C08939=1021.076,209.738,-122.791,168.989,49.902,159.469
C08940=1021.082,209.986,-122.816,168.993,49.896,159.468
C08941=1021.088,210.234,-122.842,168.996,49.891,159.468
C08942=1021.094,210.483,-122.868,169.000,49.886,159.467
C08943=1021.100,210.732,-122.894,169.003,49.880,159.467
C08944=1021.107,210.980,-122.920,169.007,49.875,159.466
C08945=1021.112,211.229,-122.946,169.010,49.869,159.465
C08946=1021.118,211.478,-122.971,169.014,49.864,159.465
C08947=1021.125,211.726,-122.997,169.017,49.858,159.464
C08948=1021.130,211.975,-123.023,169.021,49.853,159.464
C08949=1021.137,212.223,-123.049,169.024,49.848,159.463
C08950=1021.143,212.471,-123.074,169.028,49.842,159.463
C08951=1021.149,212.721,-123.101,169.032,49.837,159.462
C08952=1021.156,212.969,-123.127,169.036,49.832,159.462
C08953=1021.162,213.218,-123.152,169.039,49.826,159.461
C08954=1021.168,213.466,-123.179,169.043,49.821,159.460
C08955=1021.174,213.715,-123.204,169.046,49.816,159.460
C08956=1021.180,213.963,-123.230,169.050,49.810,159.459
C08957=1021.186,214.212,-123.256,169.053,49.805,159.459
C08958=1021.193,214.461,-123.283,169.057,49.800,159.458
C08959=1021.199,214.709,-123.308,169.060,49.794,159.457
C08960=1021.206,214.957,-123.334,169.064,49.789,159.457
C08961=1021.211,215.206,-123.360,169.068,49.784,159.457
C08962=1021.218,215.454,-123.386,169.072,49.778,159.456
C08963=1021.224,215.704,-123.412,169.075,49.773,159.455
C08964=1021.230,215.952,-123.438,169.079,49.768,159.455
C08965=1021.236,216.201,-123.464,169.082,49.763,159.454
C08966=1021.243,216.449,-123.490,169.086,49.757,159.454
C08967=1021.248,216.698,-123.516,169.089,49.752,159.453
C08968=1021.255,216.946,-123.542,169.094,49.747,159.453
C08969=1021.262,217.194,-123.568,169.097,49.742,159.452
C08970=1021.267,217.443,-123.594,169.101,49.736,159.451
C08971=1021.274,217.692,-123.620,169.104,49.731,159.451
C08972=1021.281,217.941,-123.646,169.108,49.726,159.450
C08973=1021.287,218.189,-123.672,169.111,49.721,159.450
C08974=1021.293,218.437,-123.698,169.116,49.715,159.450
C08975=1021.299,218.686,-123.725,169.119,49.711,159.449
C08976=1021.304,218.905,-123.748,169.122,49.706,159.448
C08977=1021.310,219.125,-123.771,169.126,49.701,159.448
C08978=1021.315,219.343,-123.794,169.128,49.697,159.447
C08979=1021.321,219.562,-123.818,169.132,49.692,159.447
C08980=1021.326,219.782,-123.841,169.135,49.687,159.447
C08981=1021.332,220.001,-123.864,169.138,49.683,159.446
C08982=1021.337,220.221,-123.888,169.141,49.679,159.446
C08983=1021.342,220.439,-123.911,169.144,49.674,159.445
C08984=1021.349,220.688,-123.937,169.148,49.669,159.445
C08985=1021.355,220.937,-123.963,169.152,49.664,159.444
C08986=1021.361,221.185,-123.990,169.155,49.659,159.444
C08987=1021.367,221.433,-124.016,169.159,49.654,159.443
C08988=1021.373,221.682,-124.043,169.162,49.649,159.443
C08989=1021.379,221.931,-124.070,169.167,49.644,159.442
C08990=1021.386,222.179,-124.096,169.170,49.640,159.442
C08991=1021.392,222.428,-124.123,169.173,49.635,159.441
C08992=1021.399,222.676,-124.149,169.178,49.629,159.441
C08993=1021.404,222.925,-124.175,169.181,49.624,159.440
C08994=1021.410,223.174,-124.202,169.185,49.619,159.440
C08995=1021.417,223.422,-124.228,169.188,49.614,159.439
C08996=1021.423,223.670,-124.254,169.193,49.609,159.439
C08997=1021.429,223.919,-124.281,169.196,49.604,159.438
C08998=1021.436,224.167,-124.307,169.199,49.599,159.438
C08999=1021.442,224.416,-124.334,169.204,49.595,159.438
C09000=1021.448,224.665,-124.361,169.207,49.590,159.437
C09001=1021.454,224.913,-124.387,169.211,49.584,159.437
C09002=1021.461,225.162,-124.414,169.215,49.580,159.436
C09003=1021.467,225.410,-124.440,169.218,49.575,159.435
C09004=1021.473,225.658,-124.467,169.222,49.569,159.435
C09005=1021.479,225.907,-124.494,169.226,49.565,159.435
C09006=1021.486,226.155,-124.520,169.230,49.560,159.434
C09007=1021.492,226.404,-124.547,169.233,49.555,159.434
C09008=1021.498,226.653,-124.574,169.236,49.550,159.433
C09009=1021.505,226.901,-124.600,169.241,49.545,159.433
C09010=1021.511,227.149,-124.627,169.244,49.541,159.432
C09011=1021.517,227.398,-124.654,169.249,49.535,159.432
C09012=1021.523,227.647,-124.681,169.252,49.530,159.431
C09013=1021.529,227.895,-124.708,169.255,49.526,159.431
C09014=1021.535,228.144,-124.735,169.260,49.521,159.430
C09015=1021.542,228.392,-124.762,169.263,49.516,159.430
C09016=1021.548,228.640,-124.788,169.267,49.512,159.430
C09017=1021.554,228.889,-124.815,169.271,49.507,159.429
C09018=1021.560,229.137,-124.842,169.274,49.502,159.429
C09019=1021.567,229.386,-124.869,169.278,49.497,159.428
C09020=1021.573,229.634,-124.896,169.282,49.492,159.428
C09021=1021.579,229.883,-124.923,169.286,49.488,159.427
C09022=1021.585,230.131,-124.950,169.290,49.483,159.427
C09023=1021.592,230.380,-124.977,169.293,49.479,159.427
C09024=1021.597,230.628,-125.004,169.297,49.474,159.426
C09025=1021.604,230.877,-125.032,169.301,49.469,159.426
C09026=1021.610,231.125,-125.059,169.305,49.464,159.425
C09027=1021.616,231.374,-125.086,169.308,49.460,159.425
C09028=1021.622,231.622,-125.113,169.311,49.455,159.424
C09029=1021.629,231.871,-125.140,169.316,49.451,159.424
C09030=1021.635,232.119,-125.167,169.320,49.446,159.424
C09031=1021.641,232.368,-125.194,169.323,49.441,159.423
C09032=1021.647,232.616,-125.222,169.328,49.437,159.423
C09033=1021.653,232.865,-125.249,169.331,49.432,159.422
C09034=1021.660,233.112,-125.276,169.334,49.428,159.422
C09035=1021.666,233.361,-125.303,169.339,49.423,159.422
C09036=1021.671,233.576,-125.327,169.342,49.419,159.421
C09037=1021.677,233.792,-125.350,169.345,49.415,159.421
C09038=1021.682,234.007,-125.374,169.349,49.411,159.421
C09039=1021.687,234.222,-125.397,169.351,49.407,159.420
C09040=1021.693,234.437,-125.421,169.355,49.403,159.420
C09041=1021.698,234.652,-125.444,169.358,49.399,159.420
C09042=1021.704,234.867,-125.468,169.362,49.395,159.419
C09043=1021.709,235.083,-125.492,169.365,49.391,159.419
C09044=1021.715,235.330,-125.519,169.369,49.387,159.419
C09045=1021.722,235.579,-125.547,169.373,49.382,159.418
C09046=1021.728,235.828,-125.574,169.377,49.377,159.418
C09047=1021.734,236.076,-125.601,169.380,49.373,159.417
C09048=1021.740,236.325,-125.628,169.384,49.369,159.417
C09049=1021.747,236.573,-125.656,169.388,49.364,159.417
C09050=1021.753,236.821,-125.683,169.392,49.359,159.416
C09051=1021.760,237.070,-125.710,169.396,49.355,159.416
C09052=1021.765,237.318,-125.738,169.400,49.351,159.416
C09053=1021.772,237.566,-125.766,169.404,49.346,159.415
C09054=1021.778,237.816,-125.793,169.407,49.342,159.415
C09055=1021.784,238.063,-125.820,169.412,49.337,159.414
C09056=1021.791,238.312,-125.848,169.415,49.333,159.414
C09057=1021.797,238.561,-125.875,169.419,49.329,159.414
C09058=1021.803,238.809,-125.902,169.423,49.323,159.413
C09059=1021.810,239.057,-125.930,169.427,49.319,159.413
C09060=1021.816,239.306,-125.958,169.431,49.315,159.412
C09061=1021.822,239.553,-125.986,169.435,49.310,159.412
C09062=1021.828,239.803,-126.013,169.439,49.306,159.412
C09063=1021.834,240.051,-126.041,169.442,49.302,159.412
C09064=1021.840,240.299,-126.069,169.446,49.298,159.411
C09065=1021.847,240.547,-126.096,169.451,49.293,159.411
C09066=1021.853,240.796,-126.125,169.454,49.289,159.411
C09067=1021.859,241.044,-126.152,169.458,49.285,159.410
C09068=1021.865,241.293,-126.180,169.462,49.281,159.410
C09069=1021.872,241.541,-126.208,169.466,49.276,159.410
C09070=1021.878,241.790,-126.236,169.470,49.272,159.409
C09071=1021.884,242.038,-126.264,169.474,49.268,159.409
C09072=1021.890,242.286,-126.291,169.478,49.263,159.409
C09073=1021.897,242.535,-126.319,169.482,49.259,159.408
C09074=1021.903,242.783,-126.347,169.485,49.255,159.408
C09075=1021.909,243.031,-126.375,169.489,49.251,159.407
C09076=1021.915,243.280,-126.403,169.494,49.246,159.407
C09077=1021.922,243.528,-126.431,169.497,49.242,159.407
C09078=1021.927,243.776,-126.459,169.501,49.238,159.407
C09079=1021.934,244.025,-126.487,169.505,49.233,159.406
C09080=1021.940,244.273,-126.515,169.510,49.230,159.406
C09081=1021.946,244.522,-126.544,169.513,49.225,159.406
C09082=1021.952,244.769,-126.571,169.517,49.221,159.405
C09083=1021.958,245.018,-126.600,169.520,49.217,159.405
C09084=1021.964,245.267,-126.628,169.524,49.213,159.405
C09085=1021.970,245.515,-126.656,169.529,49.209,159.405
C09086=1021.976,245.763,-126.684,169.533,49.205,159.404
C09087=1021.982,246.011,-126.713,169.536,49.200,159.404
C09088=1021.989,246.260,-126.740,169.540,49.197,159.404
C09089=1021.995,246.509,-126.769,169.545,49.192,159.403
C09090=1022.001,246.757,-126.798,169.549,49.188,159.403
C09091=1022.007,247.004,-126.825,169.553,49.185,159.403
C09092=1022.013,247.253,-126.853,169.556,49.180,159.403
C09093=1022.019,247.501,-126.883,169.561,49.176,159.402
C09094=1022.026,247.750,-126.910,169.565,49.172,159.402
C09095=1022.032,247.999,-126.939,169.569,49.168,159.402
C09096=1022.037,248.210,-126.963,169.572,49.165,159.401
C09097=1022.042,248.423,-126.987,169.576,49.161,159.401
C09098=1022.048,248.634,-127.011,169.579,49.158,159.401
C09099=1022.053,248.847,-127.036,169.583,49.155,159.401
C09100=1022.058,249.058,-127.060,169.585,49.151,159.400
C09101=1022.064,249.270,-127.084,169.589,49.147,159.400
C09102=1022.069,249.482,-127.108,169.592,49.144,159.400
C09103=1022.074,249.694,-127.132,169.596,49.141,159.400
C09104=1022.080,249.942,-127.161,169.600,49.137,159.400
C09105=1022.087,250.191,-127.190,169.604,49.133,159.399
C09106=1022.093,250.439,-127.217,169.608,49.128,159.399
C09107=1022.099,250.687,-127.246,169.612,49.125,159.399
C09108=1022.105,250.936,-127.275,169.616,49.121,159.399
C09109=1022.112,251.184,-127.303,169.620,49.117,159.398
C09110=1022.118,251.432,-127.331,169.624,49.113,159.398
C09111=1022.125,251.681,-127.361,169.629,49.109,159.398
C09112=1022.131,251.929,-127.388,169.632,49.105,159.398
C09113=1022.138,252.177,-127.417,169.636,49.101,159.397
C09114=1022.143,252.426,-127.446,169.641,49.097,159.397
C09115=1022.150,252.674,-127.474,169.645,49.093,159.397
C09116=1022.156,252.923,-127.502,169.649,49.089,159.397
C09117=1022.163,253.171,-127.531,169.653,49.086,159.396
C09118=1022.168,253.419,-127.559,169.657,49.081,159.396
C09119=1022.175,253.667,-127.588,169.661,49.078,159.396
C09120=1022.182,253.915,-127.617,169.665,49.073,159.396
C09121=1022.188,254.164,-127.646,169.669,49.070,159.395
C09122=1022.195,254.412,-127.674,169.674,49.066,159.395
C09123=1022.201,254.661,-127.702,169.678,49.062,159.395
C09124=1022.207,254.909,-127.731,169.682,49.058,159.395
C09125=1022.214,255.157,-127.760,169.685,49.054,159.394
C09126=1022.220,255.405,-127.788,169.690,49.050,159.394
C09127=1022.226,255.654,-127.817,169.694,49.046,159.394
C09128=1022.232,255.902,-127.846,169.698,49.043,159.394
C09129=1022.239,256.149,-127.875,169.702,49.039,159.394
C09130=1022.245,256.398,-127.903,169.706,49.035,159.393
C09131=1022.252,256.646,-127.932,169.710,49.031,159.393
C09132=1022.259,256.894,-127.960,169.714,49.028,159.393
C09133=1022.265,257.143,-127.989,169.719,49.023,159.393
C09134=1022.271,257.391,-128.018,169.723,49.020,159.393
C09135=1022.278,257.640,-128.047,169.727,49.016,159.392
C09136=1022.285,257.888,-128.076,169.731,49.012,159.392
C09137=1022.291,258.136,-128.105,169.736,49.008,159.392
C09138=1022.297,258.385,-128.133,169.740,49.005,159.392
C09139=1022.304,258.632,-128.162,169.743,49.000,159.391
C09140=1022.310,258.881,-128.191,169.748,48.997,159.391
C09141=1022.316,259.129,-128.220,169.752,48.993,159.391
C09142=1022.324,259.377,-128.248,169.756,48.990,159.391
C09143=1022.330,259.625,-128.277,169.760,48.985,159.391
C09144=1022.336,259.873,-128.306,169.765,48.982,159.391
C09145=1022.343,260.121,-128.335,169.769,48.978,159.390
C09146=1022.349,260.370,-128.363,169.773,48.974,159.390
C09147=1022.356,260.618,-128.393,169.777,48.971,159.390
C09148=1022.362,260.866,-128.422,169.782,48.967,159.390
C09149=1022.368,261.115,-128.452,169.786,48.964,159.390
C09150=1022.374,261.363,-128.481,169.790,48.960,159.390
C09151=1022.381,261.611,-128.510,169.794,48.957,159.389
C09152=1022.387,261.859,-128.539,169.799,48.953,159.389
C09153=1022.393,262.107,-128.568,169.803,48.949,159.389
C09154=1022.400,262.356,-128.598,169.807,48.946,159.389
C09155=1022.407,262.604,-128.627,169.811,48.942,159.389
C09156=1022.411,262.815,-128.652,169.815,48.939,159.389
C09157=1022.417,263.026,-128.677,169.818,48.936,159.389
C09158=1022.422,263.237,-128.702,169.822,48.933,159.388
C09159=1022.428,263.449,-128.727,169.826,48.930,159.388
C09160=1022.433,263.659,-128.752,169.829,48.927,159.388
C09161=1022.439,263.871,-128.777,169.833,48.924,159.388
C09162=1022.444,264.082,-128.802,169.836,48.921,159.388
C09163=1022.449,264.293,-128.827,169.841,48.918,159.388
C09164=1022.456,264.542,-128.857,169.845,48.915,159.388
C09165=1022.462,264.790,-128.886,169.849,48.911,159.387
C09166=1022.469,265.037,-128.915,169.854,48.907,159.387
C09167=1022.475,265.286,-128.945,169.858,48.904,159.387
C09168=1022.482,265.534,-128.974,169.862,48.900,159.387
C09169=1022.488,265.782,-129.004,169.866,48.897,159.387
C09170=1022.494,266.030,-129.033,169.870,48.894,159.387
C09171=1022.501,266.279,-129.063,169.875,48.890,159.387
C09172=1022.507,266.527,-129.092,169.879,48.887,159.387
C09173=1022.513,266.775,-129.122,169.883,48.883,159.386
C09174=1022.520,267.023,-129.152,169.887,48.880,159.386
C09175=1022.526,267.272,-129.181,169.892,48.876,159.386
C09176=1022.533,267.519,-129.211,169.896,48.873,159.386
C09177=1022.538,267.767,-129.241,169.900,48.869,159.386
C09178=1022.545,268.016,-129.271,169.905,48.867,159.386
C09179=1022.552,268.264,-129.300,169.909,48.863,159.386
C09180=1022.559,268.512,-129.330,169.914,48.859,159.386
C09181=1022.564,268.760,-129.360,169.918,48.856,159.386
C09182=1022.571,269.008,-129.389,169.922,48.853,159.386
C09183=1022.578,269.257,-129.419,169.926,48.849,159.385
C09184=1022.583,269.505,-129.449,169.931,48.846,159.385
C09185=1022.590,269.752,-129.479,169.935,48.843,159.385
C09186=1022.597,270.001,-129.508,169.939,48.839,159.385
C09187=1022.603,270.249,-129.539,169.944,48.836,159.385
C09188=1022.609,270.496,-129.568,169.948,48.833,159.385
C09189=1022.615,270.745,-129.598,169.953,48.830,159.385
C09190=1022.622,270.993,-129.628,169.957,48.826,159.385
C09191=1022.628,271.241,-129.659,169.961,48.824,159.385
C09192=1022.635,271.489,-129.689,169.965,48.820,159.385
C09193=1022.641,271.738,-129.719,169.971,48.817,159.385
C09194=1022.648,271.986,-129.748,169.975,48.813,159.385
C09195=1022.653,272.233,-129.779,169.979,48.811,159.385
C09196=1022.660,272.482,-129.809,169.983,48.807,159.384
C09197=1022.667,272.730,-129.838,169.988,48.804,159.384
C09198=1022.673,272.978,-129.869,169.993,48.800,159.384
C09199=1022.680,273.226,-129.898,169.997,48.798,159.384
C09200=1022.686,273.474,-129.929,170.001,48.794,159.384
C09201=1022.692,273.722,-129.959,170.005,48.791,159.384
C09202=1022.699,273.970,-129.990,170.011,48.788,159.384
C09203=1022.705,274.218,-130.020,170.015,48.785,159.384
C09204=1022.712,274.466,-130.050,170.019,48.782,159.384
C09205=1022.718,274.714,-130.080,170.023,48.779,159.384
C09206=1022.725,274.962,-130.110,170.027,48.775,159.384
C09207=1022.731,275.210,-130.141,170.033,48.772,159.384
C09208=1022.738,275.458,-130.171,170.037,48.769,159.384
C09209=1022.744,275.706,-130.201,170.041,48.766,159.384
C09210=1022.750,275.955,-130.232,170.045,48.763,159.384
C09211=1022.757,276.202,-130.262,170.051,48.760,159.384
C09212=1022.763,276.451,-130.292,170.055,48.757,159.384
C09213=1022.770,276.698,-130.322,170.059,48.754,159.384
C09214=1022.776,276.947,-130.353,170.064,48.751,159.384
C09215=1022.783,277.195,-130.383,170.069,48.748,159.384
C09216=1022.788,277.408,-130.409,170.072,48.745,159.384
C09217=1022.794,277.622,-130.435,170.077,48.742,159.384
C09218=1022.799,277.835,-130.463,170.080,48.740,159.384
C09219=1022.804,278.049,-130.489,170.084,48.737,159.384
C09220=1022.810,278.262,-130.515,170.088,48.734,159.384
C09221=1022.815,278.476,-130.541,170.091,48.733,159.384
C09222=1022.821,278.690,-130.568,170.096,48.730,159.384
C09223=1022.827,278.903,-130.595,170.099,48.727,159.384
C09224=1022.833,279.150,-130.624,170.104,48.724,159.384
C09225=1022.840,279.399,-130.655,170.109,48.721,159.384
C09226=1022.846,279.647,-130.686,170.113,48.718,159.384
C09227=1022.852,279.895,-130.717,170.117,48.716,159.384
C09228=1022.859,280.143,-130.748,170.123,48.713,159.384
C09229=1022.865,280.391,-130.777,170.127,48.710,159.384
C09230=1022.872,280.639,-130.809,170.132,48.707,159.384
C09231=1022.878,280.887,-130.839,170.136,48.703,159.384
C09232=1022.884,281.134,-130.870,170.140,48.701,159.384
C09233=1022.891,281.383,-130.901,170.145,48.697,159.384
C09234=1022.897,281.631,-130.932,170.150,48.695,159.384
C09235=1022.905,281.879,-130.963,170.154,48.692,159.384
C09236=1022.911,282.127,-130.993,170.159,48.690,159.384
C09237=1022.917,282.375,-131.025,170.164,48.686,159.384
C09238=1022.924,282.623,-131.055,170.168,48.684,159.384
C09239=1022.930,282.870,-131.086,170.173,48.681,159.384
C09240=1022.937,283.119,-131.116,170.177,48.678,159.384
C09241=1022.944,283.367,-131.148,170.182,48.675,159.384
C09242=1022.950,283.615,-131.179,170.187,48.672,159.384
C09243=1022.956,283.862,-131.210,170.191,48.669,159.384
C09244=1022.963,284.111,-131.240,170.197,48.666,159.384
C09245=1022.969,284.359,-131.272,170.201,48.663,159.384
C09246=1022.977,284.607,-131.302,170.205,48.660,159.384
C09247=1022.983,284.855,-131.333,170.210,48.658,159.384
C09248=1022.989,285.103,-131.364,170.215,48.655,159.385
C09249=1022.996,285.351,-131.395,170.220,48.652,159.385
C09250=1023.003,285.598,-131.427,170.224,48.649,159.385
C09251=1023.009,285.846,-131.458,170.228,48.647,159.385
C09252=1023.016,286.095,-131.489,170.234,48.644,159.385
C09253=1023.022,286.342,-131.520,170.238,48.641,159.385
C09254=1023.029,286.590,-131.551,170.243,48.639,159.385
C09255=1023.035,286.838,-131.583,170.248,48.636,159.385
C09256=1023.042,287.086,-131.613,170.253,48.633,159.385
C09257=1023.048,287.334,-131.645,170.257,48.630,159.385
C09258=1023.055,287.582,-131.676,170.262,48.628,159.385
C09259=1023.062,287.830,-131.708,170.266,48.625,159.385
C09260=1023.068,288.077,-131.739,170.272,48.622,159.385
C09261=1023.075,288.325,-131.770,170.276,48.620,159.386
C09262=1023.081,288.573,-131.802,170.281,48.617,159.386
C09263=1023.087,288.822,-131.833,170.285,48.615,159.386
C09264=1023.094,289.070,-131.864,170.291,48.612,159.386
C09265=1023.101,289.318,-131.896,170.295,48.609,159.386
C09266=1023.107,289.566,-131.927,170.300,48.607,159.386
C09267=1023.114,289.814,-131.959,170.304,48.604,159.386
C09268=1023.121,290.061,-131.990,170.310,48.602,159.386
C09269=1023.127,290.309,-132.022,170.314,48.599,159.386
C09270=1023.133,290.557,-132.053,170.319,48.597,159.387
C09271=1023.140,290.805,-132.085,170.324,48.594,159.387
C09272=1023.146,291.053,-132.116,170.329,48.591,159.387
C09273=1023.153,291.300,-132.148,170.333,48.589,159.387
C09274=1023.160,291.548,-132.180,170.338,48.586,159.387
C09275=1023.167,291.796,-132.211,170.343,48.583,159.387
C09276=1023.172,292.015,-132.239,170.347,48.581,159.387
C09277=1023.178,292.235,-132.267,170.352,48.579,159.387
C09278=1023.184,292.455,-132.296,170.357,48.577,159.388
C09279=1023.190,292.675,-132.323,170.360,48.575,159.388
C09280=1023.196,292.895,-132.352,170.365,48.572,159.388
C09281=1023.201,293.114,-132.380,170.369,48.570,159.388
C09282=1023.207,293.333,-132.409,170.373,48.568,159.388
C09283=1023.214,293.553,-132.436,170.378,48.566,159.388
C09284=1023.220,293.801,-132.468,170.382,48.564,159.388
C09285=1023.226,294.049,-132.500,170.388,48.561,159.388
C09286=1023.233,294.296,-132.532,170.392,48.559,159.389
C09287=1023.239,294.545,-132.564,170.397,48.557,159.389
C09288=1023.246,294.792,-132.596,170.402,48.554,159.389
C09289=1023.252,295.040,-132.629,170.408,48.552,159.389
C09290=1023.259,295.287,-132.661,170.412,48.550,159.389
C09291=1023.265,295.536,-132.693,170.417,48.547,159.389
C09292=1023.271,295.783,-132.725,170.421,48.545,159.390
C09293=1023.278,296.031,-132.757,170.427,48.542,159.390
C09294=1023.284,296.279,-132.790,170.432,48.540,159.390
C09295=1023.291,296.527,-132.821,170.436,48.538,159.390
C09296=1023.298,296.775,-132.854,170.441,48.536,159.390
C09297=1023.304,297.022,-132.887,170.447,48.533,159.391
C09298=1023.311,297.270,-132.918,170.452,48.531,159.391
C09299=1023.317,297.518,-132.951,170.456,48.529,159.391
C09300=1023.324,297.766,-132.983,170.461,48.527,159.391
C09301=1023.330,298.013,-133.015,170.467,48.524,159.392
C09302=1023.336,298.261,-133.048,170.471,48.522,159.392
C09303=1023.343,298.510,-133.080,170.476,48.520,159.392
C09304=1023.350,298.757,-133.113,170.482,48.518,159.392
C09305=1023.357,299.004,-133.145,170.486,48.516,159.392
C09306=1023.363,299.252,-133.177,170.491,48.513,159.393
C09307=1023.369,299.500,-133.209,170.496,48.511,159.393
C09308=1023.376,299.748,-133.242,170.502,48.509,159.393
C09309=1023.383,299.996,-133.275,170.506,48.507,159.393
C09310=1023.389,300.243,-133.307,170.511,48.504,159.393
C09311=1023.396,300.491,-133.339,170.517,48.502,159.394
C09312=1023.402,300.739,-133.372,170.522,48.500,159.394
C09313=1023.410,300.987,-133.404,170.526,48.498,159.394
C09314=1023.416,301.234,-133.437,170.532,48.496,159.394
C09315=1023.423,301.482,-133.470,170.537,48.494,159.395
C09316=1023.430,301.729,-133.502,170.541,48.491,159.395
C09317=1023.436,301.978,-133.535,170.547,48.489,159.395
C09318=1023.443,302.225,-133.568,170.552,48.487,159.396
C09319=1023.449,302.473,-133.599,170.557,48.485,159.396
C09320=1023.456,302.721,-133.632,170.563,48.483,159.396
C09321=1023.463,302.969,-133.664,170.567,48.481,159.396
C09322=1023.470,303.216,-133.697,170.572,48.479,159.396
C09323=1023.477,303.465,-133.730,170.578,48.477,159.397
C09324=1023.484,303.712,-133.762,170.583,48.475,159.397
C09325=1023.490,303.959,-133.795,170.587,48.472,159.397
C09326=1023.497,304.208,-133.828,170.593,48.470,159.397
C09327=1023.504,304.455,-133.860,170.598,48.468,159.398
C09328=1023.510,304.703,-133.893,170.603,48.466,159.398
C09329=1023.518,304.950,-133.926,170.609,48.464,159.398
C09330=1023.524,305.198,-133.959,170.614,48.462,159.399
C09331=1023.531,305.446,-133.992,170.619,48.460,159.399
C09332=1023.538,305.693,-134.024,170.624,48.458,159.399
C09333=1023.545,305.941,-134.057,170.629,48.456,159.399
C09334=1023.551,306.189,-134.090,170.635,48.454,159.400
C09335=1023.559,306.437,-134.123,170.640,48.452,159.400
C09336=1023.565,306.665,-134.154,170.644,48.450,159.400
C09337=1023.571,306.893,-134.183,170.649,48.448,159.400
C09338=1023.578,307.121,-134.214,170.654,48.446,159.401
C09339=1023.584,307.350,-134.244,170.659,48.444,159.401
C09340=1023.590,307.578,-134.274,170.664,48.443,159.401
C09341=1023.597,307.806,-134.305,170.669,48.440,159.401
C09342=1023.603,308.034,-134.335,170.674,48.439,159.402
C09343=1023.610,308.263,-134.365,170.678,48.437,159.402
C09344=1023.617,308.510,-134.398,170.683,48.435,159.402
C09345=1023.623,308.758,-134.431,170.689,48.433,159.403
C09346=1023.631,309.006,-134.465,170.694,48.431,159.403
C09347=1023.638,309.253,-134.497,170.700,48.429,159.404
C09348=1023.645,309.502,-134.530,170.705,48.427,159.404
C09349=1023.652,309.748,-134.563,170.711,48.425,159.404
C09350=1023.659,309.997,-134.596,170.716,48.423,159.404
C09351=1023.666,310.244,-134.630,170.722,48.421,159.405
C09352=1023.672,310.492,-134.663,170.726,48.419,159.405
C09353=1023.680,310.740,-134.697,170.731,48.418,159.405
C09354=1023.686,310.987,-134.730,170.737,48.416,159.406
C09355=1023.693,311.235,-134.763,170.742,48.414,159.406
C09356=1023.699,311.482,-134.797,170.748,48.413,159.406
C09357=1023.706,311.730,-134.831,170.754,48.411,159.407
C09358=1023.713,311.977,-134.865,170.759,48.410,159.407
C09359=1023.720,312.225,-134.898,170.763,48.407,159.407
C09360=1023.726,312.473,-134.932,170.769,48.406,159.408
C09361=1023.733,312.720,-134.966,170.774,48.404,159.408
C09362=1023.740,312.968,-134.999,170.780,48.402,159.409
C09363=1023.746,313.215,-135.034,170.785,48.401,159.409
C09364=1023.753,313.463,-135.067,170.790,48.399,159.409
C09365=1023.760,313.711,-135.100,170.797,48.397,159.410
C09366=1023.766,313.958,-135.134,170.802,48.396,159.410
C09367=1023.773,314.206,-135.168,170.808,48.394,159.411
C09368=1023.780,314.454,-135.202,170.813,48.393,159.411
C09369=1023.787,314.701,-135.236,170.818,48.391,159.411
C09370=1023.793,314.949,-135.270,170.824,48.389,159.412
C09371=1023.800,315.196,-135.304,170.829,48.388,159.412
C09372=1023.807,315.444,-135.338,170.835,48.386,159.413
C09373=1023.814,315.691,-135.371,170.840,48.384,159.413
C09374=1023.821,315.939,-135.406,170.845,48.383,159.413
C09375=1023.828,316.187,-135.439,170.851,48.381,159.414
C09376=1023.835,316.434,-135.473,170.856,48.380,159.414
C09377=1023.841,316.681,-135.507,170.862,48.378,159.415
C09378=1023.848,316.929,-135.542,170.867,48.377,159.415
C09379=1023.856,317.176,-135.576,170.873,48.375,159.416
C09380=1023.863,317.424,-135.609,170.878,48.373,159.416
C09381=1023.869,317.672,-135.644,170.884,48.372,159.417
C09382=1023.876,317.919,-135.677,170.890,48.371,159.417
C09383=1023.883,318.167,-135.711,170.896,48.369,159.418
C09384=1023.890,318.414,-135.746,170.901,48.367,159.418
C09385=1023.897,318.662,-135.780,170.906,48.366,159.418
C09386=1023.904,318.909,-135.814,170.912,48.364,159.419
C09387=1023.911,319.157,-135.848,170.917,48.363,159.419
C09388=1023.918,319.404,-135.883,170.923,48.361,159.420
C09389=1023.925,319.652,-135.917,170.928,48.360,159.420
C09390=1023.932,319.900,-135.951,170.935,48.359,159.421
C09391=1023.939,320.148,-135.985,170.940,48.357,159.421
C09392=1023.946,320.395,-136.020,170.946,48.355,159.422
C09393=1023.953,320.643,-136.054,170.951,48.354,159.422
C09394=1023.960,320.890,-136.088,170.957,48.353,159.423
C09395=1023.968,321.137,-136.122,170.963,48.351,159.423
C09396=1023.974,321.368,-136.154,170.969,48.350,159.424
C09397=1023.981,321.599,-136.186,170.974,48.348,159.424
C09398=1023.988,321.830,-136.218,170.979,48.347,159.424
C09399=1023.994,322.061,-136.250,170.984,48.346,159.425
C09400=1024.001,322.292,-136.282,170.989,48.344,159.425
C09401=1024.008,322.522,-136.315,170.994,48.343,159.426
C09402=1024.014,322.753,-136.347,171.001,48.342,159.426
C09403=1024.021,322.984,-136.378,171.006,48.340,159.427
C09404=1024.027,323.232,-136.413,171.011,48.339,159.427
C09405=1024.035,323.479,-136.447,171.017,48.338,159.428
C09406=1024.042,323.726,-136.482,171.023,48.336,159.428
C09407=1024.049,323.974,-136.516,171.028,48.335,159.429
C09408=1024.056,324.221,-136.551,171.035,48.334,159.429
C09409=1024.064,324.469,-136.585,171.040,48.332,159.430
C09410=1024.071,324.717,-136.620,171.046,48.331,159.430
C09411=1024.078,324.964,-136.655,171.052,48.330,159.431
C09412=1024.085,325.212,-136.689,171.058,48.328,159.431
C09413=1024.092,325.459,-136.724,171.064,48.327,159.432
C09414=1024.100,325.707,-136.759,171.069,48.326,159.432
C09415=1024.107,325.954,-136.794,171.075,48.324,159.433
C09416=1024.114,326.202,-136.828,171.081,48.323,159.433
C09417=1024.122,326.449,-136.862,171.087,48.322,159.434
C09418=1024.129,326.697,-136.898,171.093,48.320,159.434
C09419=1024.137,326.944,-136.932,171.098,48.320,159.435
C09420=1024.144,327.191,-136.967,171.105,48.318,159.436
C09421=1024.151,327.438,-137.002,171.110,48.317,159.436
C09422=1024.158,327.686,-137.037,171.116,48.316,159.437
C09423=1024.165,327.934,-137.072,171.123,48.314,159.437
C09424=1024.172,328.181,-137.108,171.128,48.314,159.438
C09425=1024.180,328.428,-137.142,171.134,48.312,159.438
C09426=1024.186,328.675,-137.177,171.140,48.311,159.439
C09427=1024.194,328.923,-137.213,171.146,48.310,159.440
C09428=1024.200,329.171,-137.248,171.152,48.309,159.440
C09429=1024.208,329.418,-137.282,171.158,48.308,159.441
C09430=1024.216,329.665,-137.319,171.164,48.307,159.441
C09431=1024.222,329.913,-137.354,171.170,48.306,159.442
C09432=1024.229,330.160,-137.389,171.176,48.305,159.443
C09433=1024.237,330.408,-137.424,171.182,48.304,159.443
C09434=1024.244,330.655,-137.459,171.188,48.303,159.444
C09435=1024.251,330.902,-137.495,171.194,48.302,159.444
C09436=1024.258,331.150,-137.530,171.200,48.300,159.445
C09437=1024.265,331.397,-137.565,171.206,48.300,159.446
C09438=1024.273,331.645,-137.602,171.212,48.298,159.446
C09439=1024.280,331.892,-137.636,171.218,48.297,159.447
C09440=1024.288,332.140,-137.672,171.224,48.297,159.448
C09441=1024.295,332.387,-137.708,171.231,48.296,159.448
C09442=1024.302,332.634,-137.743,171.236,48.295,159.449
C09443=1024.309,332.881,-137.779,171.242,48.294,159.449
C09444=1024.317,333.128,-137.813,171.249,48.292,159.450
C09445=1024.324,333.377,-137.849,171.255,48.292,159.451
C09446=1024.331,333.623,-137.885,171.261,48.291,159.451
C09447=1024.339,333.871,-137.921,171.267,48.290,159.452
C09448=1024.346,334.118,-137.956,171.273,48.290,159.453
C09449=1024.353,334.366,-137.992,171.279,48.288,159.453
C09450=1024.360,334.612,-138.028,171.286,48.287,159.454
C09451=1024.368,334.860,-138.064,171.292,48.287,159.455
C09452=1024.375,335.107,-138.100,171.298,48.286,159.455
C09453=1024.383,335.355,-138.136,171.304,48.285,159.456
C09454=1024.390,335.603,-138.171,171.311,48.284,159.457
C09455=1024.396,335.850,-138.208,171.316,48.283,159.457
C09456=1024.404,336.078,-138.240,171.323,48.282,159.458
C09457=1024.411,336.307,-138.274,171.328,48.282,159.459
C09458=1024.417,336.535,-138.307,171.334,48.281,159.459
C09459=1024.424,336.764,-138.341,171.339,48.280,159.460
C09460=1024.431,336.993,-138.374,171.346,48.279,159.461
C09461=1024.438,337.221,-138.407,171.351,48.279,159.461
C09462=1024.444,337.450,-138.440,171.357,48.278,159.462
C09463=1024.451,337.678,-138.474,171.363,48.277,159.463
C09464=1024.459,337.926,-138.510,171.369,48.277,159.463
C09465=1024.466,338.172,-138.546,171.375,48.276,159.464
C09466=1024.473,338.420,-138.582,171.382,48.275,159.465
C09467=1024.481,338.668,-138.618,171.389,48.274,159.466
C09468=1024.489,338.915,-138.654,171.394,48.274,159.466
C09469=1024.496,339.162,-138.690,171.401,48.273,159.467
C09470=1024.503,339.409,-138.727,171.407,48.272,159.468
C09471=1024.511,339.657,-138.764,171.414,48.272,159.469
C09472=1024.518,339.904,-138.800,171.420,48.271,159.469
C09473=1024.526,340.151,-138.836,171.426,48.270,159.470
C09474=1024.533,340.398,-138.872,171.433,48.270,159.471
C09475=1024.540,340.646,-138.909,171.440,48.269,159.472
C09476=1024.548,340.893,-138.946,171.446,48.268,159.472
C09477=1024.555,341.140,-138.981,171.452,48.268,159.473
C09478=1024.563,341.387,-139.018,171.459,48.268,159.474
C09479=1024.570,341.635,-139.054,171.465,48.267,159.475
C09480=1024.578,341.882,-139.091,171.472,48.266,159.475
C09481=1024.585,342.129,-139.128,171.478,48.265,159.476
C09482=1024.593,342.376,-139.165,171.484,48.265,159.477
C09483=1024.600,342.623,-139.201,171.491,48.264,159.478
C09484=1024.607,342.870,-139.237,171.497,48.264,159.479
C09485=1024.615,343.118,-139.275,171.504,48.263,159.479
C09486=1024.622,343.365,-139.311,171.511,48.263,159.480
C09487=1024.630,343.612,-139.348,171.517,48.262,159.481
C09488=1024.637,343.860,-139.385,171.524,48.262,159.482
C09489=1024.645,344.106,-139.422,171.530,48.262,159.483
C09490=1024.652,344.354,-139.458,171.537,48.261,159.484
C09491=1024.660,344.601,-139.495,171.544,48.261,159.484
C09492=1024.668,344.848,-139.532,171.550,48.260,159.485
C09493=1024.675,345.096,-139.569,171.557,48.259,159.486
C09494=1024.683,345.342,-139.606,171.563,48.259,159.487
C09495=1024.690,345.590,-139.644,171.570,48.259,159.488
C09496=1024.698,345.837,-139.680,171.577,48.259,159.489
C09497=1024.706,346.084,-139.717,171.583,48.258,159.489
C09498=1024.713,346.331,-139.754,171.590,48.257,159.490
C09499=1024.721,346.578,-139.791,171.597,48.257,159.491
C09500=1024.728,346.825,-139.828,171.604,48.257,159.492
C09501=1024.736,347.072,-139.865,171.610,48.256,159.493
C09502=1024.743,347.319,-139.902,171.618,48.256,159.494
C09503=1024.751,347.566,-139.939,171.624,48.256,159.495
C09504=1024.760,347.814,-139.977,171.631,48.255,159.495
C09505=1024.767,348.061,-140.014,171.637,48.255,159.496
C09506=1024.774,348.308,-140.052,171.644,48.255,159.497
C09507=1024.782,348.555,-140.089,171.651,48.255,159.498
C09508=1024.790,348.802,-140.126,171.657,48.254,159.499
C09509=1024.798,349.049,-140.163,171.664,48.254,159.500
C09510=1024.805,349.296,-140.201,171.671,48.254,159.501
C09511=1024.813,349.544,-140.239,171.678,48.254,159.502
C09512=1024.821,349.791,-140.275,171.685,48.253,159.503
C09513=1024.828,350.038,-140.313,171.692,48.253,159.504
C09514=1024.836,350.284,-140.351,171.699,48.253,159.505
C09515=1024.843,350.531,-140.388,171.706,48.253,159.505
C09516=1024.851,350.759,-140.423,171.712,48.253,159.506
C09517=1024.858,350.986,-140.458,171.718,48.252,159.507
C09518=1024.864,351.213,-140.492,171.724,48.253,159.508
C09519=1024.872,351.440,-140.528,171.731,48.252,159.509
C09520=1024.878,351.667,-140.562,171.737,48.252,159.510
C09521=1024.886,351.894,-140.597,171.744,48.252,159.511
C09522=1024.893,352.121,-140.631,171.751,48.252,159.512
C09523=1024.900,352.348,-140.666,171.757,48.252,159.512
C09524=1024.908,352.595,-140.703,171.764,48.252,159.513
C09525=1024.916,352.842,-140.741,171.771,48.252,159.514
C09526=1024.924,353.089,-140.779,171.778,48.252,159.515
C09527=1024.932,353.335,-140.817,171.784,48.251,159.516
C09528=1024.940,353.583,-140.855,171.791,48.251,159.517
C09529=1024.947,353.830,-140.893,171.799,48.251,159.518
C09530=1024.956,354.077,-140.930,171.806,48.251,159.519
C09531=1024.963,354.324,-140.968,171.814,48.251,159.520
C09532=1024.971,354.572,-141.006,171.821,48.251,159.521
C09533=1024.979,354.818,-141.044,171.828,48.251,159.522
C09534=1024.987,355.064,-141.082,171.835,48.251,159.523
C09535=1024.995,355.312,-141.120,171.842,48.251,159.524
C09536=1025.002,355.559,-141.158,171.849,48.251,159.525
C09537=1025.011,355.806,-141.197,171.856,48.251,159.526
C09538=1025.018,356.052,-141.235,171.863,48.251,159.527
C09539=1025.026,356.300,-141.274,171.870,48.251,159.528
C09540=1025.034,356.547,-141.311,171.877,48.252,159.530
C09541=1025.042,356.794,-141.350,171.884,48.252,159.531
C09542=1025.049,357.041,-141.388,171.892,48.251,159.532
C09543=1025.058,357.287,-141.426,171.899,48.251,159.533
C09544=1025.066,357.535,-141.465,171.906,48.251,159.534
C09545=1025.074,357.781,-141.503,171.914,48.252,159.535
C09546=1025.082,358.028,-141.542,171.921,48.252,159.536
C09547=1025.090,358.275,-141.580,171.928,48.252,159.537
C09548=1025.098,358.522,-141.618,171.936,48.252,159.538
C09549=1025.106,358.769,-141.657,171.943,48.252,159.539
C09550=1025.113,359.016,-141.695,171.950,48.252,159.540
C09551=1025.122,359.263,-141.734,171.958,48.253,159.541
C09552=1025.130,359.510,-141.773,171.965,48.253,159.542
C09553=1025.138,359.756,-141.811,171.973,48.253,159.544
C09554=1025.146,360.003,-141.850,171.980,48.253,159.545
C09555=1025.154,360.251,-141.889,171.987,48.253,159.546
C09556=1025.162,360.497,-141.928,171.995,48.254,159.547
C09557=1025.170,360.744,-141.966,172.002,48.255,159.548
C09558=1025.178,360.991,-142.005,172.010,48.254,159.549
C09559=1025.186,361.238,-142.044,172.017,48.255,159.550
C09560=1025.194,361.485,-142.083,172.024,48.255,159.551
C09561=1025.202,361.731,-142.122,172.032,48.255,159.553
C09562=1025.210,361.978,-142.161,172.040,48.256,159.554
C09563=1025.218,362.225,-142.200,172.048,48.256,159.555
C09564=1025.226,362.472,-142.239,172.055,48.256,159.556
C09565=1025.234,362.719,-142.279,172.062,48.257,159.557
C09566=1025.242,362.965,-142.318,172.070,48.257,159.559
C09567=1025.250,363.212,-142.356,172.078,48.258,159.560
C09568=1025.259,363.459,-142.396,172.085,48.258,159.561
C09569=1025.266,363.706,-142.436,172.092,48.259,159.562
C09570=1025.275,363.953,-142.474,172.101,48.259,159.563
C09571=1025.283,364.199,-142.513,172.108,48.259,159.564
C09572=1025.291,364.446,-142.553,172.115,48.260,159.566
C09573=1025.300,364.693,-142.591,172.124,48.260,159.567
C09574=1025.307,364.940,-142.631,172.131,48.261,159.568
C09575=1025.316,365.187,-142.671,172.138,48.262,159.569
C09576=1025.323,365.417,-142.707,172.145,48.262,159.570
C09577=1025.331,365.647,-142.744,172.153,48.262,159.571
C09578=1025.338,365.878,-142.781,172.160,48.263,159.573
C09579=1025.346,366.108,-142.818,172.168,48.263,159.574
C09580=1025.355,366.338,-142.854,172.175,48.264,159.575
C09581=1025.362,366.568,-142.891,172.182,48.264,159.576
C09582=1025.370,366.799,-142.928,172.189,48.265,159.577
C09583=1025.378,367.030,-142.965,172.197,48.265,159.578
C09584=1025.386,367.276,-143.004,172.205,48.265,159.580
C09585=1025.394,367.523,-143.044,172.212,48.266,159.581
C09586=1025.403,367.769,-143.084,172.221,48.267,159.582
C09587=1025.411,368.016,-143.123,172.229,48.267,159.584
C09588=1025.420,368.262,-143.163,172.236,48.268,159.585
C09589=1025.428,368.510,-143.203,172.244,48.268,159.586
C09590=1025.437,368.757,-143.242,172.252,48.270,159.588
C09591=1025.445,369.003,-143.283,172.260,48.270,159.589
C09592=1025.453,369.250,-143.322,172.268,48.271,159.590
C09593=1025.461,369.496,-143.362,172.277,48.271,159.591
C09594=1025.470,369.742,-143.402,172.284,48.272,159.593
C09595=1025.478,369.990,-143.443,172.293,48.273,159.594
C09596=1025.487,370.236,-143.483,172.300,48.273,159.595
C09597=1025.494,370.483,-143.523,172.309,48.274,159.597
C09598=1025.502,370.729,-143.563,172.316,48.275,159.598
C09599=1025.512,370.976,-143.604,172.325,48.276,159.599
C09600=1025.519,371.223,-143.643,172.333,48.277,159.601
C09601=1025.528,371.469,-143.684,172.341,48.277,159.602
C09602=1025.536,371.716,-143.723,172.349,48.278,159.604
C09603=1025.545,371.962,-143.764,172.357,48.279,159.605
C09604=1025.553,372.209,-143.804,172.365,48.280,159.606
C09605=1025.561,372.455,-143.845,172.373,48.281,159.608
C09606=1025.570,372.702,-143.885,172.382,48.282,159.609
C09607=1025.578,372.948,-143.925,172.390,48.283,159.611
C09608=1025.588,373.195,-143.966,172.398,48.283,159.612
C09609=1025.596,373.441,-144.006,172.406,48.284,159.613
C09610=1025.605,373.688,-144.047,172.415,48.285,159.615
C09611=1025.613,373.934,-144.088,172.423,48.286,159.616
C09612=1025.621,374.181,-144.128,172.431,48.287,159.618
C09613=1025.630,374.428,-144.168,172.440,48.288,159.619
C09614=1025.638,374.674,-144.208,172.449,48.289,159.620
C09615=1025.648,374.921,-144.249,172.456,48.290,159.622
C09616=1025.657,375.167,-144.291,172.465,48.291,159.623
C09617=1025.665,375.413,-144.331,172.474,48.292,159.625
C09618=1025.674,375.660,-144.372,172.481,48.293,159.626
C09619=1025.682,375.907,-144.412,172.490,48.294,159.628
C09620=1025.691,376.153,-144.453,172.499,48.295,159.629
C09621=1025.700,376.400,-144.494,172.508,48.296,159.631
C09622=1025.709,376.646,-144.534,172.515,48.297,159.632
C09623=1025.718,376.893,-144.575,172.524,48.298,159.633
C09624=1025.726,377.140,-144.616,172.533,48.299,159.635
C09625=1025.734,377.386,-144.657,172.542,48.300,159.637
C09626=1025.743,377.632,-144.699,172.550,48.301,159.638
C09627=1025.751,377.878,-144.739,172.559,48.303,159.640
C09628=1025.761,378.125,-144.781,172.567,48.303,159.641
C09629=1025.770,378.372,-144.822,172.576,48.304,159.643
C09630=1025.779,378.618,-144.863,172.584,48.306,159.644
C09631=1025.787,378.864,-144.905,172.593,48.307,159.646
C09632=1025.796,379.111,-144.946,172.602,48.308,159.647
C09633=1025.804,379.357,-144.987,172.611,48.309,159.649
C09634=1025.813,379.603,-145.029,172.620,48.311,159.651
C09635=1025.821,379.850,-145.070,172.627,48.312,159.652
C09636=1025.830,380.091,-145.111,172.637,48.313,159.654
C09637=1025.839,380.332,-145.151,172.645,48.314,159.655
C09638=1025.848,380.573,-145.191,172.654,48.315,159.657
C09639=1025.857,380.814,-145.232,172.662,48.317,159.658
C09640=1025.865,381.055,-145.272,172.671,48.318,159.660
C09641=1025.874,381.296,-145.313,172.680,48.319,159.661
C09642=1025.882,381.537,-145.354,172.689,48.320,159.663
C09643=1025.891,381.778,-145.395,172.697,48.322,159.665
C09644=1025.900,382.025,-145.437,172.706,48.323,159.666
C09645=1025.909,382.271,-145.479,172.715,48.325,159.668
C09646=1025.918,382.517,-145.520,172.724,48.326,159.669
C09647=1025.927,382.764,-145.562,172.733,48.327,159.671
C09648=1025.937,383.010,-145.603,172.742,48.329,159.673
C09649=1025.946,383.256,-145.645,172.751,48.330,159.674
C09650=1025.955,383.503,-145.687,172.760,48.331,159.676
C09651=1025.964,383.748,-145.729,172.769,48.333,159.678
C09652=1025.973,383.995,-145.771,172.778,48.334,159.679
C09653=1025.982,384.241,-145.812,172.787,48.336,159.681
C09654=1025.991,384.487,-145.854,172.796,48.337,159.683
C09655=1026.000,384.733,-145.897,172.805,48.339,159.684
C09656=1026.009,384.980,-145.938,172.814,48.340,159.686
C09657=1026.018,385.227,-145.980,172.825,48.342,159.688
C09658=1026.028,385.472,-146.023,172.834,48.343,159.690
C09659=1026.036,385.719,-146.065,172.843,48.344,159.691
C09660=1026.046,385.964,-146.107,172.852,48.346,159.693
C09661=1026.055,386.211,-146.149,172.861,48.348,159.695
C09662=1026.064,386.457,-146.191,172.871,48.349,159.697
C09663=1026.073,386.704,-146.233,172.880,48.351,159.698
C09664=1026.083,386.949,-146.276,172.889,48.353,159.700
C09665=1026.092,387.195,-146.318,172.899,48.354,159.702
C09666=1026.101,387.442,-146.361,172.909,48.356,159.704
C09667=1026.110,387.688,-146.403,172.918,48.357,159.705
C09668=1026.119,387.934,-146.446,172.927,48.359,159.707
C09669=1026.129,388.180,-146.488,172.936,48.361,159.709
C09670=1026.138,388.426,-146.531,172.946,48.362,159.711
C09671=1026.147,388.672,-146.574,172.956,48.364,159.713
C09672=1026.157,388.919,-146.617,172.965,48.366,159.714
C09673=1026.166,389.164,-146.659,172.974,48.368,159.716
C09674=1026.176,389.411,-146.702,172.984,48.370,159.718
C09675=1026.184,389.657,-146.745,172.994,48.371,159.720
C09676=1026.194,389.903,-146.788,173.003,48.373,159.722
C09677=1026.203,390.149,-146.830,173.013,48.375,159.724
C09678=1026.212,390.395,-146.873,173.023,48.376,159.726
C09679=1026.222,390.641,-146.917,173.033,48.378,159.728
C09680=1026.231,390.887,-146.959,173.042,48.380,159.729
C09681=1026.240,391.133,-147.003,173.052,48.382,159.731
C09682=1026.250,391.379,-147.046,173.062,48.384,159.733
C09683=1026.260,391.625,-147.088,173.071,48.386,159.735
C09684=1026.269,391.872,-147.132,173.082,48.388,159.737
C09685=1026.278,392.117,-147.175,173.091,48.390,159.739
C09686=1026.288,392.363,-147.218,173.100,48.391,159.741
C09687=1026.298,392.609,-147.262,173.111,48.393,159.743
C09688=1026.307,392.855,-147.304,173.120,48.395,159.745
C09689=1026.317,393.101,-147.348,173.131,48.397,159.747
C09690=1026.326,393.348,-147.391,173.140,48.399,159.749
C09691=1026.336,393.593,-147.434,173.151,48.401,159.751
C09692=1026.345,393.839,-147.479,173.160,48.403,159.752
C09693=1026.355,394.085,-147.522,173.171,48.405,159.755
C09694=1026.364,394.332,-147.565,173.181,48.407,159.757
C09695=1026.373,394.577,-147.609,173.191,48.409,159.759
C09696=1026.384,394.849,-147.657,173.202,48.412,159.761
C09697=1026.395,395.122,-147.705,173.213,48.414,159.763
C09698=1026.406,395.394,-147.754,173.225,48.416,159.765
C09699=1026.416,395.666,-147.802,173.236,48.418,159.768
C09700=1026.426,395.912,-147.847,173.245,48.421,159.770
C09701=1026.436,396.158,-147.890,173.256,48.423,159.772
C09702=1026.445,396.404,-147.934,173.267,48.425,159.774
C09703=1026.456,396.650,-147.978,173.276,48.427,159.776
C09704=1026.465,396.896,-148.022,173.287,48.429,159.778
C09705=1026.475,397.142,-148.066,173.298,48.431,159.780
C09706=1026.485,397.388,-148.110,173.307,48.434,159.782
C09707=1026.494,397.634,-148.154,173.318,48.436,159.784
C09708=1026.504,397.879,-148.198,173.329,48.438,159.786
C09709=1026.514,398.125,-148.243,173.339,48.441,159.788
C09710=1026.524,398.371,-148.286,173.349,48.443,159.791
C09711=1026.534,398.617,-148.331,173.360,48.445,159.793
C09712=1026.543,398.863,-148.375,173.371,48.447,159.795
C09713=1026.554,399.108,-148.419,173.381,48.450,159.797
C09714=1026.563,399.354,-148.463,173.392,48.452,159.799
C09715=1026.573,399.600,-148.509,173.402,48.454,159.801
C09716=1026.584,399.845,-148.553,173.413,48.456,159.803
C09717=1026.593,400.092,-148.597,173.423,48.459,159.806
C09718=1026.603,400.337,-148.642,173.434,48.461,159.808
C09719=1026.613,400.583,-148.686,173.445,48.464,159.810
C09720=1026.622,400.828,-148.731,173.456,48.466,159.812
C09721=1026.633,401.074,-148.776,173.467,48.469,159.815
C09722=1026.643,401.320,-148.821,173.477,48.471,159.817
C09723=1026.652,401.566,-148.865,173.488,48.474,159.819
C09724=1026.663,401.812,-148.910,173.498,48.476,159.821
C09725=1026.673,402.057,-148.956,173.510,48.479,159.824
C09726=1026.683,402.302,-149.000,173.520,48.481,159.826
C09727=1026.693,402.549,-149.046,173.531,48.484,159.828
C09728=1026.703,402.794,-149.090,173.543,48.486,159.830
C09729=1026.712,403.040,-149.135,173.554,48.489,159.833
C09730=1026.723,403.285,-149.180,173.564,48.491,159.835
C09731=1026.733,403.530,-149.225,173.576,48.494,159.837
C09732=1026.744,403.777,-149.271,173.587,48.497,159.840
C09733=1026.753,404.022,-149.315,173.598,48.499,159.842
C09734=1026.764,404.268,-149.361,173.609,48.502,159.844
C09735=1026.774,404.513,-149.406,173.620,48.505,159.847
C09736=1026.784,404.759,-149.452,173.631,48.508,159.849
C09737=1026.794,405.004,-149.497,173.642,48.510,159.851
C09738=1026.805,405.250,-149.543,173.654,48.513,159.854
C09739=1026.815,405.496,-149.588,173.666,48.515,159.856
C09740=1026.825,405.741,-149.633,173.677,48.518,159.859
C09741=1026.835,405.987,-149.679,173.688,48.521,159.861
C09742=1026.846,406.233,-149.725,173.699,48.524,159.863
C09743=1026.856,406.478,-149.770,173.710,48.526,159.866
C09744=1026.867,406.723,-149.816,173.723,48.529,159.868
C09745=1026.877,406.969,-149.861,173.734,48.532,159.871
C09746=1026.888,407.215,-149.907,173.745,48.535,159.873
C09747=1026.898,407.461,-149.953,173.756,48.538,159.876
C09748=1026.908,407.706,-149.999,173.769,48.540,159.878
C09749=1026.919,407.951,-150.044,173.780,48.543,159.881
C09750=1026.929,408.197,-150.090,173.791,48.546,159.883
C09751=1026.940,408.442,-150.136,173.804,48.549,159.886
C09752=1026.951,408.688,-150.182,173.815,48.552,159.888
C09753=1026.961,408.934,-150.228,173.826,48.555,159.891
C09754=1026.972,409.179,-150.274,173.838,48.557,159.893
C09755=1026.983,409.425,-150.320,173.850,48.561,159.896
C09756=1026.995,409.709,-150.374,173.864,48.564,159.899
C09757=1027.008,409.995,-150.428,173.878,48.568,159.902
C09758=1027.020,410.281,-150.482,173.892,48.571,159.905
C09759=1027.032,410.566,-150.535,173.905,48.575,159.908
C09760=1027.043,410.811,-150.582,173.918,48.578,159.910
C09761=1027.053,411.057,-150.628,173.929,48.581,159.913
C09762=1027.064,411.303,-150.675,173.942,48.584,159.916
C09763=1027.075,411.548,-150.722,173.953,48.587,159.918
C09764=1027.086,411.793,-150.768,173.966,48.590,159.921
C09765=1027.097,412.038,-150.815,173.978,48.593,159.924
C09766=1027.107,412.284,-150.862,173.990,48.597,159.926
C09767=1027.118,412.529,-150.909,174.002,48.600,159.929
C09768=1027.129,412.774,-150.955,174.014,48.603,159.931
C09769=1027.139,413.020,-151.002,174.027,48.606,159.934
C09770=1027.151,413.266,-151.049,174.039,48.609,159.937
C09771=1027.162,413.511,-151.095,174.051,48.613,159.940
C09772=1027.172,413.756,-151.143,174.064,48.616,159.942
C09773=1027.183,414.002,-151.190,174.077,48.619,159.945
C09774=1027.195,414.246,-151.237,174.089,48.622,159.948
C09775=1027.206,414.492,-151.285,174.101,48.626,159.951
C09776=1027.216,414.737,-151.331,174.114,48.629,159.954
C09777=1027.228,414.983,-151.378,174.126,48.632,159.956
C09778=1027.239,415.228,-151.425,174.139,48.636,159.959
C09779=1027.250,415.473,-151.473,174.152,48.639,159.962
C09780=1027.261,415.718,-151.520,174.165,48.642,159.965
C09781=1027.272,415.964,-151.567,174.178,48.646,159.968
C09782=1027.284,416.209,-151.615,174.190,48.650,159.971
C09783=1027.294,416.454,-151.662,174.202,48.653,159.973
C09784=1027.306,416.699,-151.710,174.215,48.656,159.976
C09785=1027.317,416.945,-151.758,174.228,48.660,159.979
C09786=1027.328,417.190,-151.805,174.241,48.663,159.982
C09787=1027.339,417.435,-151.853,174.254,48.667,159.985
C09788=1027.351,417.680,-151.901,174.267,48.671,159.988
C09789=1027.362,417.925,-151.949,174.280,48.674,159.991
C09790=1027.372,418.170,-151.997,174.293,48.677,159.994
C09791=1027.384,418.415,-152.045,174.307,48.681,159.997
C09792=1027.395,418.661,-152.093,174.320,48.684,160.000
C09793=1027.407,418.906,-152.141,174.333,48.688,160.003
C09794=1027.418,419.151,-152.189,174.346,48.692,160.006
C09795=1027.430,419.396,-152.237,174.359,48.696,160.009
C09796=1027.441,419.650,-152.287,174.374,48.699,160.012
C09797=1027.453,419.904,-152.337,174.387,48.703,160.015
C09798=1027.465,420.158,-152.387,174.401,48.707,160.018
C09799=1027.477,420.412,-152.437,174.414,48.711,160.021
C09800=1027.488,420.658,-152.485,174.428,48.714,160.024
C09801=1027.500,420.903,-152.533,174.442,48.718,160.027
C09802=1027.511,421.147,-152.582,174.455,48.722,160.030
C09803=1027.523,421.393,-152.630,174.469,48.726,160.034
C09804=1027.535,421.637,-152.679,174.482,48.730,160.037
C09805=1027.546,421.883,-152.727,174.497,48.733,160.040
C09806=1027.559,422.128,-152.776,174.510,48.737,160.043
C09807=1027.570,422.373,-152.824,174.524,48.741,160.046
C09808=1027.582,422.619,-152.873,174.538,48.745,160.049
C09809=1027.593,422.863,-152.922,174.552,48.749,160.053
C09810=1027.605,423.108,-152.971,174.566,48.753,160.056
C09811=1027.617,423.352,-153.020,174.580,48.757,160.059
C09812=1027.629,423.598,-153.069,174.593,48.761,160.062
C09813=1027.640,423.843,-153.118,174.608,48.765,160.065
C09814=1027.651,424.087,-153.167,174.621,48.769,160.069
C09815=1027.664,424.333,-153.216,174.635,48.772,160.072
C09816=1027.679,424.637,-153.277,174.653,48.778,160.076
C09817=1027.694,424.943,-153.339,174.671,48.783,160.080
C09818=1027.708,425.247,-153.401,174.689,48.788,160.084
C09819=1027.723,425.551,-153.461,174.706,48.793,160.088
C09820=1027.735,425.797,-153.511,174.721,48.797,160.092
C09821=1027.748,426.042,-153.561,174.735,48.801,160.095
C09822=1027.759,426.286,-153.610,174.750,48.805,160.099
C09823=1027.771,426.531,-153.660,174.765,48.809,160.102
C09824=1027.783,426.777,-153.709,174.780,48.814,160.106
C09825=1027.795,427.021,-153.759,174.794,48.818,160.109
C09826=1027.807,427.266,-153.809,174.809,48.822,160.112
C09827=1027.820,427.510,-153.859,174.823,48.827,160.116
C09828=1027.832,427.755,-153.909,174.837,48.831,160.119
C09829=1027.844,427.999,-153.959,174.852,48.835,160.123
C09830=1027.856,428.244,-154.009,174.868,48.839,160.126
C09831=1027.868,428.489,-154.059,174.883,48.844,160.130
C09832=1027.881,428.734,-154.109,174.898,48.848,160.133
C09833=1027.893,428.979,-154.160,174.913,48.852,160.137
C09834=1027.905,429.223,-154.210,174.928,48.857,160.140
C09835=1027.918,429.468,-154.260,174.943,48.861,160.144
C09836=1027.930,429.712,-154.311,174.958,48.866,160.148
C09837=1027.943,429.957,-154.361,174.974,48.870,160.151
C09838=1027.955,430.202,-154.411,174.989,48.875,160.155
C09839=1027.968,430.446,-154.462,175.004,48.879,160.158
C09840=1027.980,430.691,-154.512,175.020,48.883,160.162
C09841=1027.992,430.936,-154.563,175.035,48.888,160.166
C09842=1028.004,431.180,-154.614,175.050,48.892,160.169
C09843=1028.017,431.425,-154.664,175.066,48.897,160.173
C09844=1028.029,431.669,-154.715,175.081,48.902,160.177
C09845=1028.043,431.914,-154.766,175.097,48.906,160.180
C09846=1028.055,432.158,-154.817,175.112,48.911,160.184
C09847=1028.067,432.403,-154.867,175.128,48.915,160.188
C09848=1028.081,432.648,-154.918,175.144,48.920,160.192
C09849=1028.093,432.892,-154.969,175.160,48.924,160.195
C09850=1028.107,433.137,-155.020,175.176,48.929,160.199
C09851=1028.119,433.381,-155.071,175.191,48.934,160.203
C09852=1028.133,433.625,-155.123,175.208,48.939,160.207
C09853=1028.145,433.870,-155.174,175.224,48.943,160.211
C09854=1028.157,434.114,-155.225,175.239,48.948,160.215
C09855=1028.171,434.358,-155.277,175.256,48.953,160.218
C09856=1028.184,434.603,-155.328,175.272,48.958,160.222
C09857=1028.197,434.847,-155.380,175.289,48.962,160.226
C09858=1028.209,435.092,-155.431,175.305,48.967,160.230
C09859=1028.222,435.336,-155.483,175.321,48.972,160.234
C09860=1028.235,435.580,-155.534,175.337,48.977,160.238
C09861=1028.249,435.825,-155.586,175.353,48.982,160.242
C09862=1028.261,436.069,-155.638,175.370,48.987,160.246
C09863=1028.275,436.313,-155.690,175.387,48.992,160.250
C09864=1028.288,436.557,-155.742,175.403,48.997,160.254
C09865=1028.301,436.802,-155.794,175.420,49.002,160.258
C09866=1028.314,437.045,-155.846,175.438,49.007,160.262
C09867=1028.327,437.290,-155.898,175.454,49.011,160.266
C09868=1028.340,437.534,-155.950,175.471,49.016,160.270
C09869=1028.354,437.779,-156.002,175.488,49.021,160.274
C09870=1028.368,438.022,-156.055,175.504,49.027,160.279
C09871=1028.381,438.266,-156.107,175.522,49.031,160.283
C09872=1028.394,438.511,-156.159,175.539,49.037,160.287
C09873=1028.408,438.755,-156.212,175.556,49.042,160.291
C09874=1028.421,438.999,-156.264,175.574,49.047,160.295
C09875=1028.434,439.243,-156.317,175.591,49.053,160.300
C09876=1028.450,439.510,-156.374,175.610,49.058,160.304
C09877=1028.464,439.776,-156.432,175.629,49.064,160.309
C09878=1028.479,440.042,-156.490,175.648,49.069,160.314
C09879=1028.493,440.309,-156.547,175.667,49.075,160.318
C09880=1028.507,440.553,-156.600,175.685,49.080,160.323
C09881=1028.521,440.797,-156.653,175.703,49.086,160.327
C09882=1028.534,441.041,-156.706,175.720,49.091,160.331
C09883=1028.549,441.285,-156.759,175.738,49.097,160.336
C09884=1028.562,441.528,-156.813,175.757,49.102,160.340
C09885=1028.576,441.772,-156.865,175.775,49.107,160.345
C09886=1028.590,442.017,-156.919,175.792,49.113,160.349
C09887=1028.604,442.260,-156.972,175.810,49.118,160.353
C09888=1028.618,442.503,-157.025,175.828,49.123,160.358
C09889=1028.632,442.746,-157.078,175.847,49.129,160.362
C09890=1028.647,442.990,-157.132,175.865,49.134,160.367
C09891=1028.660,443.234,-157.184,175.883,49.140,160.371
C09892=1028.675,443.476,-157.237,175.901,49.145,160.376
C09893=1028.691,443.720,-157.289,175.920,49.150,160.380
C09894=1028.707,443.964,-157.341,175.939,49.155,160.385
C09895=1028.724,444.207,-157.392,175.957,49.160,160.389
C09896=1028.740,444.451,-157.442,175.976,49.165,160.394
C09897=1028.758,444.694,-157.493,175.995,49.170,160.398
C09898=1028.775,444.939,-157.543,176.014,49.175,160.403
C09899=1028.794,445.183,-157.593,176.033,49.180,160.407
C09900=1028.813,445.427,-157.642,176.052,49.184,160.411
C09901=1028.832,445.671,-157.691,176.072,49.189,160.416
C09902=1028.852,445.915,-157.739,176.091,49.193,160.420
C09903=1028.872,446.160,-157.787,176.110,49.198,160.425
C09904=1028.893,446.404,-157.835,176.130,49.202,160.429
C09905=1028.914,446.648,-157.882,176.149,49.207,160.433
C09906=1028.935,446.893,-157.929,176.169,49.211,160.438
C09907=1028.958,447.137,-157.975,176.188,49.215,160.442
C09908=1028.980,447.382,-158.021,176.208,49.219,160.447
C09909=1029.003,447.626,-158.066,176.227,49.223,160.451
C09910=1029.027,447.871,-158.111,176.247,49.227,160.455
C09911=1029.051,448.116,-158.156,176.268,49.231,160.460
C09912=1029.076,448.361,-158.201,176.288,49.235,160.464
C09913=1029.100,448.606,-158.245,176.308,49.239,160.468
C09914=1029.126,448.851,-158.289,176.329,49.242,160.473
C09915=1029.152,449.095,-158.332,176.348,49.246,160.477
C09916=1029.178,449.340,-158.375,176.369,49.250,160.482
C09917=1029.205,449.587,-158.417,176.390,49.253,160.486
C09918=1029.232,449.831,-158.459,176.411,49.256,160.490
C09919=1029.260,450.076,-158.501,176.431,49.260,160.495
C09920=1029.289,450.321,-158.542,176.452,49.264,160.499
C09921=1029.317,450.567,-158.583,176.473,49.267,160.503
C09922=1029.346,450.813,-158.624,176.494,49.270,160.508
C09923=1029.376,451.058,-158.663,176.515,49.273,160.512
C09924=1029.406,451.303,-158.703,176.536,49.276,160.516
C09925=1029.437,451.549,-158.742,176.558,49.279,160.521
C09926=1029.468,451.794,-158.780,176.579,49.282,160.525
C09927=1029.500,452.040,-158.819,176.601,49.285,160.529
C09928=1029.532,452.286,-158.856,176.622,49.288,160.534
C09929=1029.565,452.532,-158.894,176.644,49.291,160.538
C09930=1029.598,452.777,-158.932,176.666,49.294,160.542
C09931=1029.631,453.023,-158.968,176.687,49.296,160.546
C09932=1029.666,453.269,-159.004,176.709,49.299,160.551
C09933=1029.700,453.515,-159.040,176.731,49.301,160.555
C09934=1029.735,453.761,-159.076,176.754,49.304,160.559
C09935=1029.770,454.005,-159.111,176.775,49.307,160.564
C09936=1029.493,454.078,-159.446,176.779,49.368,160.584
C09937=1029.457,453.833,-159.411,176.756,49.366,160.580
C09938=1029.422,453.587,-159.375,176.734,49.364,160.575
C09939=1029.388,453.341,-159.339,176.712,49.361,160.571
C09940=1029.353,453.095,-159.303,176.690,49.359,160.567
C09941=1029.320,452.850,-159.267,176.668,49.356,160.562
C09942=1029.287,452.605,-159.230,176.646,49.353,160.558
C09943=1029.253,452.358,-159.192,176.625,49.350,160.554
C09944=1029.221,452.112,-159.155,176.602,49.348,160.549
C09945=1029.190,451.867,-159.116,176.581,49.345,160.545
C09946=1029.158,451.622,-159.078,176.560,49.342,160.541
C09947=1029.127,451.376,-159.039,176.538,49.339,160.536
C09948=1029.096,451.130,-159.000,176.517,49.336,160.532
C09949=1029.066,450.885,-158.960,176.496,49.333,160.528
C09950=1029.038,450.640,-158.920,176.475,49.330,160.523
C09951=1029.009,450.395,-158.879,176.454,49.327,160.519
C09952=1028.980,450.149,-158.838,176.433,49.324,160.515
C09953=1028.952,449.903,-158.796,176.413,49.321,160.511
C09954=1028.924,449.659,-158.755,176.392,49.317,160.506
C09955=1028.898,449.413,-158.713,176.371,49.313,160.502
C09956=1028.871,449.168,-158.670,176.350,49.310,160.497
C09957=1028.845,448.923,-158.627,176.330,49.307,160.493
C09958=1028.819,448.678,-158.584,176.310,49.303,160.489
C09959=1028.794,448.433,-158.540,176.289,49.299,160.484
C09960=1028.769,448.188,-158.496,176.269,49.296,160.480
C09961=1028.745,447.943,-158.451,176.248,49.292,160.476
C09962=1028.722,447.698,-158.406,176.228,49.288,160.471
C09963=1028.699,447.454,-158.361,176.209,49.284,160.467
C09964=1028.675,447.209,-158.315,176.189,49.280,160.462
C09965=1028.654,446.965,-158.268,176.169,49.276,160.458
C09966=1028.631,446.720,-158.222,176.150,49.272,160.454
C09967=1028.610,446.475,-158.175,176.130,49.268,160.449
C09968=1028.589,446.232,-158.127,176.110,49.264,160.445
C09969=1028.568,445.987,-158.079,176.091,49.259,160.441
C09970=1028.548,445.743,-158.031,176.072,49.254,160.436
C09971=1028.529,445.499,-157.982,176.052,49.251,160.432
C09972=1028.510,445.255,-157.933,176.033,49.246,160.427
C09973=1028.492,445.010,-157.884,176.014,49.241,160.423
C09974=1028.473,444.766,-157.835,175.995,49.236,160.418
C09975=1028.456,444.523,-157.784,175.976,49.231,160.414
C09976=1028.439,444.280,-157.733,175.957,49.227,160.410
C09977=1028.422,444.035,-157.683,175.938,49.222,160.405
C09978=1028.406,443.791,-157.631,175.920,49.217,160.401
C09979=1028.390,443.548,-157.579,175.901,49.212,160.396
C09980=1028.375,443.306,-157.527,175.883,49.207,160.392
C09981=1028.360,443.062,-157.474,175.865,49.202,160.387
C09982=1028.346,442.819,-157.421,175.846,49.196,160.383
C09983=1028.332,442.576,-157.368,175.828,49.191,160.378
C09984=1028.318,442.332,-157.315,175.810,49.186,160.374
C09985=1028.303,442.088,-157.261,175.792,49.180,160.369
C09986=1028.290,441.845,-157.209,175.773,49.175,160.365
C09987=1028.276,441.600,-157.155,175.755,49.170,160.361
C09988=1028.262,441.357,-157.102,175.737,49.165,160.356
C09989=1028.249,441.113,-157.049,175.720,49.159,160.352
C09990=1028.234,440.869,-156.996,175.702,49.154,160.347
C09991=1028.220,440.625,-156.943,175.684,49.149,160.343
C09992=1028.207,440.381,-156.890,175.666,49.144,160.339
C09993=1028.193,440.124,-156.834,175.647,49.138,160.334
C09994=1028.178,439.867,-156.779,175.629,49.133,160.330
C09995=1028.164,439.609,-156.723,175.611,49.127,160.325
C09996=1028.150,439.352,-156.667,175.592,49.122,160.321
//INST
///DATE 2021/06/17 10:59
///ATTR SC,RW,RJ
////FRAME ROBOT
///GROUP1 RB1
NOP
MOVL C00000 V=800.0 PL=0
MOVL C00001 V=800.0 PL=0
MOVL C00002 V=800.0 PL=0
MOVL C00003 V=800.0 PL=0
MOVL C00004 V=800.0 PL=0
MOVL C00005 V=800.0 PL=0
MOVL C00006 V=800.0 PL=0
MOVL C00007 V=800.0 PL=0
MOVL C00008 V=800.0 PL=0
MOVL C00009 V=800.0 PL=0
MOVL C00010 V=800.0 PL=0
MOVL C00011 V=800.0 PL=0
MOVL C00012 V=800.0 PL=0
MOVL C00013 V=800.0 PL=0
MOVL C00014 V=800.0 PL=0
MOVL C00015 V=800.0 PL=0
MOVL C00016 V=800.0 PL=0
MOVL C00017 V=800.0 PL=0
MOVL C00018 V=800.0 PL=0
MOVL C00019 V=800.0 PL=0
MOVL C00020 V=800.0 PL=0
MOVL C00021 V=800.0 PL=0
MOVL C00022 V=800.0 PL=0
MOVL C00023 V=800.0 PL=0
MOVL C00024 V=800.0 PL=0
MOVL C00025 V=800.0 PL=0
MOVL C00026 V=800.0 PL=0
MOVL C00027 V=800.0 PL=0
MOVL C00028 V=800.0 PL=0
MOVL C00029 V=800.0 PL=0
MOVL C00030 V=800.0 PL=0
MOVL C00031 V=800.0 PL=0
MOVL C00032 V=800.0 PL=0
MOVL C00033 V=800.0 PL=0
MOVL C00034 V=800.0 PL=0
MOVL C00035 V=800.0 PL=0
MOVL C00036 V=800.0 PL=0
MOVL C00037 V=800.0 PL=0
MOVL C00038 V=800.0 PL=0
MOVL C00039 V=800.0 PL=0
MOVL C00040 V=800.0 PL=0
MOVL C00041 V=800.0 PL=0
MOVL C00042 V=800.0 PL=0
MOVL C00043 V=800.0 PL=0
MOVL C00044 V=800.0 PL=0
MOVL C00045 V=800.0 PL=0
MOVL C00046 V=800.0 PL=0
MOVL C00047 V=800.0 PL=0
MOVL C00048 V=800.0 PL=0
MOVL C00049 V=800.0 PL=0
MOVL C00050 V=800.0 PL=0
MOVL C00051 V=800.0 PL=0
MOVL C00052 V=800.0 PL=0
MOVL C00053 V=800.0 PL=0
MOVL C00054 V=800.0 PL=0
MOVL C00055 V=800.0 PL=0
MOVL C00056 V=800.0 PL=0
MOVL C00057 V=800.0 PL=0
MOVL C00058 V=800.0 PL=0
MOVL C00059 V=800.0 PL=0
MOVL C00060 V=800.0 PL=0
MOVL C00061 V=800.0 PL=0
MOVL C00062 V=800.0 PL=0
MOVL C00063 V=800.0 PL=0
MOVL C00064 V=800.0 PL=0
MOVL C00065 V=800.0 PL=0
MOVL C00066 V=800.0 PL=0
MOVL C00067 V=800.0 PL=0
MOVL C00068 V=800.0 PL=0
MOVL C00069 V=800.0 PL=0
MOVL C00070 V=800.0 PL=0
MOVL C00071 V=800.0 PL=0
MOVL C00072 V=800.0 PL=0
MOVL C00073 V=800.0 PL=0
MOVL C00074 V=800.0 PL=0
MOVL C00075 V=800.0 PL=0
MOVL C00076 V=800.0 PL=0
MOVL C00077 V=800.0 PL=0
MOVL C00078 V=800.0 PL=0
MOVL C00079 V=800.0 PL=0
MOVL C00080 V=800.0 PL=0
MOVL C00081 V=800.0 PL=0
MOVL C00082 V=800.0 PL=0
MOVL C00083 V=800.0 PL=0
MOVL C00084 V=800.0 PL=0
MOVL C00085 V=800.0 PL=0
MOVL C00086 V=800.0 PL=0
MOVL C00087 V=800.0 PL=0
MOVL C00088 V=800.0 PL=0
MOVL C00089 V=800.0 PL=0
MOVL C00090 V=800.0 PL=0
MOVL C00091 V=800.0 PL=0
MOVL C00092 V=800.0 PL=0
MOVL C00093 V=800.0 PL=0
MOVL C00094 V=800.0 PL=0
MOVL C00095 V=800.0 PL=0
MOVL C00096 V=800.0 PL=0
MOVL C00097 V=800.0 PL=0
MOVL C00098 V=800.0 PL=0
MOVL C00099 V=800.0 PL=0
MOVL C00100 V=800.0 PL=0
MOVL C00101 V=800.0 PL=0
MOVL C00102 V=800.0 PL=0
MOVL C00103 V=800.0 PL=0
MOVL C00104 V=800.0 PL=0
MOVL C00105 V=800.0 PL=0
MOVL C00106 V=800.0 PL=0
MOVL C00107 V=800.0 PL=0
MOVL C00108 V=800.0 PL=0
MOVL C00109 V=800.0 PL=0
MOVL C00110 V=800.0 PL=0
MOVL C00111 V=800.0 PL=0
MOVL C00112 V=800.0 PL=0
MOVL C00113 V=800.0 PL=0
MOVL C00114 V=800.0 PL=0
MOVL C00115 V=800.0 PL=0
MOVL C00116 V=800.0 PL=0
MOVL C00117 V=800.0 PL=0
MOVL C00118 V=800.0 PL=0
MOVL C00119 V=800.0 PL=0
MOVL C00120 V=800.0 PL=0
MOVL C00121 V=800.0 PL=0
MOVL C00122 V=800.0 PL=0
MOVL C00123 V=800.0 PL=0
MOVL C00124 V=800.0 PL=0
MOVL C00125 V=800.0 PL=0
MOVL C00126 V=800.0 PL=0
MOVL C00127 V=800.0 PL=0
MOVL C00128 V=800.0 PL=0
MOVL C00129 V=800.0 PL=0
MOVL C00130 V=800.0 PL=0
MOVL C00131 V=800.0 PL=0
MOVL C00132 V=800.0 PL=0
MOVL C00133 V=800.0 PL=0
MOVL C00134 V=800.0 PL=0
MOVL C00135 V=800.0 PL=0
MOVL C00136 V=800.0 PL=0
MOVL C00137 V=800.0 PL=0
MOVL C00138 V=800.0 PL=0
MOVL C00139 V=800.0 PL=0
MOVL C00140 V=800.0 PL=0
MOVL C00141 V=800.0 PL=0
MOVL C00142 V=800.0 PL=0
MOVL C00143 V=800.0 PL=0
MOVL C00144 V=800.0 PL=0
MOVL C00145 V=800.0 PL=0
MOVL C00146 V=800.0 PL=0
MOVL C00147 V=800.0 PL=0
MOVL C00148 V=800.0 PL=0
MOVL C00149 V=800.0 PL=0
MOVL C00150 V=800.0 PL=0
MOVL C00151 V=800.0 PL=0
MOVL C00152 V=800.0 PL=0
MOVL C00153 V=800.0 PL=0
MOVL C00154 V=800.0 PL=0
MOVL C00155 V=800.0 PL=0
MOVL C00156 V=800.0 PL=0
MOVL C00157 V=800.0 PL=0
MOVL C00158 V=800.0 PL=0
MOVL C00159 V=800.0 PL=0
MOVL C00160 V=800.0 PL=0
MOVL C00161 V=800.0 PL=0
MOVL C00162 V=800.0 PL=0
MOVL C00163 V=800.0 PL=0
MOVL C00164 V=800.0 PL=0
MOVL C00165 V=800.0 PL=0
MOVL C00166 V=800.0 PL=0
MOVL C00167 V=800.0 PL=0
MOVL C00168 V=800.0 PL=0
MOVL C00169 V=800.0 PL=0
MOVL C00170 V=800.0 PL=0
MOVL C00171 V=800.0 PL=0
MOVL C00172 V=800.0 PL=0
MOVL C00173 V=800.0 PL=0
MOVL C00174 V=800.0 PL=0
MOVL C00175 V=800.0 PL=0
MOVL C00176 V=800.0 PL=0
MOVL C00177 V=800.0 PL=0
MOVL C00178 V=800.0 PL=0
MOVL C00179 V=800.0 PL=0
MOVL C00180 V=800.0 PL=0
MOVL C00181 V=800.0 PL=0
MOVL C00182 V=800.0 PL=0
MOVL C00183 V=800.0 PL=0
MOVL C00184 V=800.0 PL=0
MOVL C00185 V=800.0 PL=0
MOVL C00186 V=800.0 PL=0
MOVL C00187 V=800.0 PL=0
MOVL C00188 V=800.0 PL=0
MOVL C00189 V=800.0 PL=0
MOVL C00190 V=800.0 PL=0
MOVL C00191 V=800.0 PL=0
MOVL C00192 V=800.0 PL=0
MOVL C00193 V=800.0 PL=0
MOVL C00194 V=800.0 PL=0
MOVL C00195 V=800.0 PL=0
MOVL C00196 V=800.0 PL=0
MOVL C00197 V=800.0 PL=0
MOVL C00198 V=800.0 PL=0
MOVL C00199 V=800.0 PL=0
MOVL C00200 V=800.0 PL=0
MOVL C00201 V=800.0 PL=0
MOVL C00202 V=800.0 PL=0
MOVL C00203 V=800.0 PL=0
MOVL C00204 V=800.0 PL=0
MOVL C00205 V=800.0 PL=0
MOVL C00206 V=800.0 PL=0
MOVL C00207 V=800.0 PL=0
MOVL C00208 V=800.0 PL=0
MOVL C00209 V=800.0 PL=0
MOVL C00210 V=800.0 PL=0
MOVL C00211 V=800.0 PL=0
MOVL C00212 V=800.0 PL=0
MOVL C00213 V=800.0 PL=0
MOVL C00214 V=800.0 PL=0
MOVL C00215 V=800.0 PL=0
MOVL C00216 V=800.0 PL=0
MOVL C00217 V=800.0 PL=0
MOVL C00218 V=800.0 PL=0
MOVL C00219 V=800.0 PL=0
MOVL C00220 V=800.0 PL=0
MOVL C00221 V=800.0 PL=0
MOVL C00222 V=800.0 PL=0
MOVL C00223 V=800.0 PL=0
MOVL C00224 V=800.0 PL=0
MOVL C00225 V=800.0 PL=0
MOVL C00226 V=800.0 PL=0
MOVL C00227 V=800.0 PL=0
MOVL C00228 V=800.0 PL=0
MOVL C00229 V=800.0 PL=0
MOVL C00230 V=800.0 PL=0
MOVL C00231 V=800.0 PL=0
MOVL C00232 V=800.0 PL=0
MOVL C00233 V=800.0 PL=0
MOVL C00234 V=800.0 PL=0
MOVL C00235 V=800.0 PL=0
MOVL C00236 V=800.0 PL=0
MOVL C00237 V=800.0 PL=0
MOVL C00238 V=800.0 PL=0
MOVL C00239 V=800.0 PL=0
MOVL C00240 V=800.0 PL=0
MOVL C00241 V=800.0 PL=0
MOVL C00242 V=800.0 PL=0
MOVL C00243 V=800.0 PL=0
MOVL C00244 V=800.0 PL=0
MOVL C00245 V=800.0 PL=0
MOVL C00246 V=800.0 PL=0
MOVL C00247 V=800.0 PL=0
MOVL C00248 V=800.0 PL=0
MOVL C00249 V=800.0 PL=0
MOVL C00250 V=800.0 PL=0
MOVL C00251 V=800.0 PL=0
MOVL C00252 V=800.0 PL=0
MOVL C00253 V=800.0 PL=0
MOVL C00254 V=800.0 PL=0
MOVL C00255 V=800.0 PL=0
MOVL C00256 V=800.0 PL=0
MOVL C00257 V=800.0 PL=0
MOVL C00258 V=800.0 PL=0
MOVL C00259 V=800.0 PL=0
MOVL C00260 V=800.0 PL=0
MOVL C00261 V=800.0 PL=0
MOVL C00262 V=800.0 PL=0
MOVL C00263 V=800.0 PL=0
MOVL C00264 V=800.0 PL=0
MOVL C00265 V=800.0 PL=0
MOVL C00266 V=800.0 PL=0
MOVL C00267 V=800.0 PL=0
MOVL C00268 V=800.0 PL=0
MOVL C00269 V=800.0 PL=0
MOVL C00270 V=800.0 PL=0
MOVL C00271 V=800.0 PL=0
MOVL C00272 V=800.0 PL=0
MOVL C00273 V=800.0 PL=0
MOVL C00274 V=800.0 PL=0
MOVL C00275 V=800.0 PL=0
MOVL C00276 V=800.0 PL=0
MOVL C00277 V=800.0 PL=0
MOVL C00278 V=800.0 PL=0
MOVL C00279 V=800.0 PL=0
MOVL C00280 V=800.0 PL=0
MOVL C00281 V=800.0 PL=0
MOVL C00282 V=800.0 PL=0
MOVL C00283 V=800.0 PL=0
MOVL C00284 V=800.0 PL=0
MOVL C00285 V=800.0 PL=0
MOVL C00286 V=800.0 PL=0
MOVL C00287 V=800.0 PL=0
MOVL C00288 V=800.0 PL=0
MOVL C00289 V=800.0 PL=0
MOVL C00290 V=800.0 PL=0
MOVL C00291 V=800.0 PL=0
MOVL C00292 V=800.0 PL=0
MOVL C00293 V=800.0 PL=0
MOVL C00294 V=800.0 PL=0
MOVL C00295 V=800.0 PL=0
MOVL C00296 V=800.0 PL=0
MOVL C00297 V=800.0 PL=0
MOVL C00298 V=800.0 PL=0
MOVL C00299 V=800.0 PL=0
MOVL C00300 V=800.0 PL=0
MOVL C00301 V=800.0 PL=0
MOVL C00302 V=800.0 PL=0
MOVL C00303 V=800.0 PL=0
MOVL C00304 V=800.0 PL=0
MOVL C00305 V=800.0 PL=0
MOVL C00306 V=800.0 PL=0
MOVL C00307 V=800.0 PL=0
MOVL C00308 V=800.0 PL=0
MOVL C00309 V=800.0 PL=0
MOVL C00310 V=800.0 PL=0
MOVL C00311 V=800.0 PL=0
MOVL C00312 V=800.0 PL=0
MOVL C00313 V=800.0 PL=0
MOVL C00314 V=800.0 PL=0
MOVL C00315 V=800.0 PL=0
MOVL C00316 V=800.0 PL=0
MOVL C00317 V=800.0 PL=0
MOVL C00318 V=800.0 PL=0
MOVL C00319 V=800.0 PL=0
MOVL C00320 V=800.0 PL=0
MOVL C00321 V=800.0 PL=0
MOVL C00322 V=800.0 PL=0
MOVL C00323 V=800.0 PL=0
MOVL C00324 V=800.0 PL=0
MOVL C00325 V=800.0 PL=0
MOVL C00326 V=800.0 PL=0
MOVL C00327 V=800.0 PL=0
MOVL C00328 V=800.0 PL=0
MOVL C00329 V=800.0 PL=0
MOVL C00330 V=800.0 PL=0
MOVL C00331 V=800.0 PL=0
MOVL C00332 V=800.0 PL=0
MOVL C00333 V=800.0 PL=0
MOVL C00334 V=800.0 PL=0
MOVL C00335 V=800.0 PL=0
MOVL C00336 V=800.0 PL=0
MOVL C00337 V=800.0 PL=0
MOVL C00338 V=800.0 PL=0
MOVL C00339 V=800.0 PL=0
MOVL C00340 V=800.0 PL=0
MOVL C00341 V=800.0 PL=0
MOVL C00342 V=800.0 PL=0
MOVL C00343 V=800.0 PL=0
MOVL C00344 V=800.0 PL=0
MOVL C00345 V=800.0 PL=0
MOVL C00346 V=800.0 PL=0
MOVL C00347 V=800.0 PL=0
MOVL C00348 V=800.0 PL=0
MOVL C00349 V=800.0 PL=0
MOVL C00350 V=800.0 PL=0
MOVL C00351 V=800.0 PL=0
MOVL C00352 V=800.0 PL=0
MOVL C00353 V=800.0 PL=0
MOVL C00354 V=800.0 PL=0
MOVL C00355 V=800.0 PL=0
MOVL C00356 V=800.0 PL=0
MOVL C00357 V=800.0 PL=0
MOVL C00358 V=800.0 PL=0
MOVL C00359 V=800.0 PL=0
MOVL C00360 V=800.0 PL=0
MOVL C00361 V=800.0 PL=0
MOVL C00362 V=800.0 PL=0
MOVL C00363 V=800.0 PL=0
MOVL C00364 V=800.0 PL=0
MOVL C00365 V=800.0 PL=0
MOVL C00366 V=800.0 PL=0
MOVL C00367 V=800.0 PL=0
MOVL C00368 V=800.0 PL=0
MOVL C00369 V=800.0 PL=0
MOVL C00370 V=800.0 PL=0
MOVL C00371 V=800.0 PL=0
MOVL C00372 V=800.0 PL=0
MOVL C00373 V=800.0 PL=0
MOVL C00374 V=800.0 PL=0
MOVL C00375 V=800.0 PL=0
MOVL C00376 V=800.0 PL=0
MOVL C00377 V=800.0 PL=0
MOVL C00378 V=800.0 PL=0
MOVL C00379 V=800.0 PL=0
MOVL C00380 V=800.0 PL=0
MOVL C00381 V=800.0 PL=0
MOVL C00382 V=800.0 PL=0
MOVL C00383 V=800.0 PL=0
MOVL C00384 V=800.0 PL=0
MOVL C00385 V=800.0 PL=0
MOVL C00386 V=800.0 PL=0
MOVL C00387 V=800.0 PL=0
MOVL C00388 V=800.0 PL=0
MOVL C00389 V=800.0 PL=0
MOVL C00390 V=800.0 PL=0
MOVL C00391 V=800.0 PL=0
MOVL C00392 V=800.0 PL=0
MOVL C00393 V=800.0 PL=0
MOVL C00394 V=800.0 PL=0
MOVL C00395 V=800.0 PL=0
MOVL C00396 V=800.0 PL=0
MOVL C00397 V=800.0 PL=0
MOVL C00398 V=800.0 PL=0
MOVL C00399 V=800.0 PL=0
MOVL C00400 V=800.0 PL=0
MOVL C00401 V=800.0 PL=0
MOVL C00402 V=800.0 PL=0
MOVL C00403 V=800.0 PL=0
MOVL C00404 V=800.0 PL=0
MOVL C00405 V=800.0 PL=0
MOVL C00406 V=800.0 PL=0
MOVL C00407 V=800.0 PL=0
MOVL C00408 V=800.0 PL=0
MOVL C00409 V=800.0 PL=0
MOVL C00410 V=800.0 PL=0
MOVL C00411 V=800.0 PL=0
MOVL C00412 V=800.0 PL=0
MOVL C00413 V=800.0 PL=0
MOVL C00414 V=800.0 PL=0
MOVL C00415 V=800.0 PL=0
MOVL C00416 V=800.0 PL=0
MOVL C00417 V=800.0 PL=0
MOVL C00418 V=800.0 PL=0
MOVL C00419 V=800.0 PL=0
MOVL C00420 V=800.0 PL=0
MOVL C00421 V=800.0 PL=0
MOVL C00422 V=800.0 PL=0
MOVL C00423 V=800.0 PL=0
MOVL C00424 V=800.0 PL=0
MOVL C00425 V=800.0 PL=0
MOVL C00426 V=800.0 PL=0
MOVL C00427 V=800.0 PL=0
MOVL C00428 V=800.0 PL=0
MOVL C00429 V=800.0 PL=0
MOVL C00430 V=800.0 PL=0
MOVL C00431 V=800.0 PL=0
MOVL C00432 V=800.0 PL=0
MOVL C00433 V=800.0 PL=0
MOVL C00434 V=800.0 PL=0
MOVL C00435 V=800.0 PL=0
MOVL C00436 V=800.0 PL=0
MOVL C00437 V=800.0 PL=0
MOVL C00438 V=800.0 PL=0
MOVL C00439 V=800.0 PL=0
MOVL C00440 V=800.0 PL=0
MOVL C00441 V=800.0 PL=0
MOVL C00442 V=800.0 PL=0
MOVL C00443 V=800.0 PL=0
MOVL C00444 V=800.0 PL=0
MOVL C00445 V=800.0 PL=0
MOVL C00446 V=800.0 PL=0
MOVL C00447 V=800.0 PL=0
MOVL C00448 V=800.0 PL=0
MOVL C00449 V=800.0 PL=0
MOVL C00450 V=800.0 PL=0
MOVL C00451 V=800.0 PL=0
MOVL C00452 V=800.0 PL=0
MOVL C00453 V=800.0 PL=0
MOVL C00454 V=800.0 PL=0
MOVL C00455 V=800.0 PL=0
MOVL C00456 V=800.0 PL=0
MOVL C00457 V=800.0 PL=0
MOVL C00458 V=800.0 PL=0
MOVL C00459 V=800.0 PL=0
MOVL C00460 V=800.0 PL=0
MOVL C00461 V=800.0 PL=0
MOVL C00462 V=800.0 PL=0
MOVL C00463 V=800.0 PL=0
MOVL C00464 V=800.0 PL=0
MOVL C00465 V=800.0 PL=0
MOVL C00466 V=800.0 PL=0
MOVL C00467 V=800.0 PL=0
MOVL C00468 V=800.0 PL=0
MOVL C00469 V=800.0 PL=0
MOVL C00470 V=800.0 PL=0
MOVL C00471 V=800.0 PL=0
MOVL C00472 V=800.0 PL=0
MOVL C00473 V=800.0 PL=0
MOVL C00474 V=800.0 PL=0
MOVL C00475 V=800.0 PL=0
MOVL C00476 V=800.0 PL=0
MOVL C00477 V=800.0 PL=0
MOVL C00478 V=800.0 PL=0
MOVL C00479 V=800.0 PL=0
MOVL C00480 V=800.0 PL=0
MOVL C00481 V=800.0 PL=0
MOVL C00482 V=800.0 PL=0
MOVL C00483 V=800.0 PL=0
MOVL C00484 V=800.0 PL=0
MOVL C00485 V=800.0 PL=0
MOVL C00486 V=800.0 PL=0
MOVL C00487 V=800.0 PL=0
MOVL C00488 V=800.0 PL=0
MOVL C00489 V=800.0 PL=0
MOVL C00490 V=800.0 PL=0
MOVL C00491 V=800.0 PL=0
MOVL C00492 V=800.0 PL=0
MOVL C00493 V=800.0 PL=0
MOVL C00494 V=800.0 PL=0
MOVL C00495 V=800.0 PL=0
MOVL C00496 V=800.0 PL=0
MOVL C00497 V=800.0 PL=0
MOVL C00498 V=800.0 PL=0
MOVL C00499 V=800.0 PL=0
MOVL C00500 V=800.0 PL=0
MOVL C00501 V=800.0 PL=0
MOVL C00502 V=800.0 PL=0
MOVL C00503 V=800.0 PL=0
MOVL C00504 V=800.0 PL=0
MOVL C00505 V=800.0 PL=0
MOVL C00506 V=800.0 PL=0
MOVL C00507 V=800.0 PL=0
MOVL C00508 V=800.0 PL=0
MOVL C00509 V=800.0 PL=0
MOVL C00510 V=800.0 PL=0
MOVL C00511 V=800.0 PL=0
MOVL C00512 V=800.0 PL=0
MOVL C00513 V=800.0 PL=0
MOVL C00514 V=800.0 PL=0
MOVL C00515 V=800.0 PL=0
MOVL C00516 V=800.0 PL=0
MOVL C00517 V=800.0 PL=0
MOVL C00518 V=800.0 PL=0
MOVL C00519 V=800.0 PL=0
MOVL C00520 V=800.0 PL=0
MOVL C00521 V=800.0 PL=0
MOVL C00522 V=800.0 PL=0
MOVL C00523 V=800.0 PL=0
MOVL C00524 V=800.0 PL=0
MOVL C00525 V=800.0 PL=0
MOVL C00526 V=800.0 PL=0
MOVL C00527 V=800.0 PL=0
MOVL C00528 V=800.0 PL=0
MOVL C00529 V=800.0 PL=0
MOVL C00530 V=800.0 PL=0
MOVL C00531 V=800.0 PL=0
MOVL C00532 V=800.0 PL=0
MOVL C00533 V=800.0 PL=0
MOVL C00534 V=800.0 PL=0
MOVL C00535 V=800.0 PL=0
MOVL C00536 V=800.0 PL=0
MOVL C00537 V=800.0 PL=0
MOVL C00538 V=800.0 PL=0
MOVL C00539 V=800.0 PL=0
MOVL C00540 V=800.0 PL=0
MOVL C00541 V=800.0 PL=0
MOVL C00542 V=800.0 PL=0
MOVL C00543 V=800.0 PL=0
MOVL C00544 V=800.0 PL=0
MOVL C00545 V=800.0 PL=0
MOVL C00546 V=800.0 PL=0
MOVL C00547 V=800.0 PL=0
MOVL C00548 V=800.0 PL=0
MOVL C00549 V=800.0 PL=0
MOVL C00550 V=800.0 PL=0
MOVL C00551 V=800.0 PL=0
MOVL C00552 V=800.0 PL=0
MOVL C00553 V=800.0 PL=0
MOVL C00554 V=800.0 PL=0
MOVL C00555 V=800.0 PL=0
MOVL C00556 V=800.0 PL=0
MOVL C00557 V=800.0 PL=0
MOVL C00558 V=800.0 PL=0
MOVL C00559 V=800.0 PL=0
MOVL C00560 V=800.0 PL=0
MOVL C00561 V=800.0 PL=0
MOVL C00562 V=800.0 PL=0
MOVL C00563 V=800.0 PL=0
MOVL C00564 V=800.0 PL=0
MOVL C00565 V=800.0 PL=0
MOVL C00566 V=800.0 PL=0
MOVL C00567 V=800.0 PL=0
MOVL C00568 V=800.0 PL=0
MOVL C00569 V=800.0 PL=0
MOVL C00570 V=800.0 PL=0
MOVL C00571 V=800.0 PL=0
MOVL C00572 V=800.0 PL=0
MOVL C00573 V=800.0 PL=0
MOVL C00574 V=800.0 PL=0
MOVL C00575 V=800.0 PL=0
MOVL C00576 V=800.0 PL=0
MOVL C00577 V=800.0 PL=0
MOVL C00578 V=800.0 PL=0
MOVL C00579 V=800.0 PL=0
MOVL C00580 V=800.0 PL=0
MOVL C00581 V=800.0 PL=0
MOVL C00582 V=800.0 PL=0
MOVL C00583 V=800.0 PL=0
MOVL C00584 V=800.0 PL=0
MOVL C00585 V=800.0 PL=0
MOVL C00586 V=800.0 PL=0
MOVL C00587 V=800.0 PL=0
MOVL C00588 V=800.0 PL=0
MOVL C00589 V=800.0 PL=0
MOVL C00590 V=800.0 PL=0
MOVL C00591 V=800.0 PL=0
MOVL C00592 V=800.0 PL=0
MOVL C00593 V=800.0 PL=0
MOVL C00594 V=800.0 PL=0
MOVL C00595 V=800.0 PL=0
MOVL C00596 V=800.0 PL=0
MOVL C00597 V=800.0 PL=0
MOVL C00598 V=800.0 PL=0
MOVL C00599 V=800.0 PL=0
MOVL C00600 V=800.0 PL=0
MOVL C00601 V=800.0 PL=0
MOVL C00602 V=800.0 PL=0
MOVL C00603 V=800.0 PL=0
MOVL C00604 V=800.0 PL=0
MOVL C00605 V=800.0 PL=0
MOVL C00606 V=800.0 PL=0
MOVL C00607 V=800.0 PL=0
MOVL C00608 V=800.0 PL=0
MOVL C00609 V=800.0 PL=0
MOVL C00610 V=800.0 PL=0
MOVL C00611 V=800.0 PL=0
MOVL C00612 V=800.0 PL=0
MOVL C00613 V=800.0 PL=0
MOVL C00614 V=800.0 PL=0
MOVL C00615 V=800.0 PL=0
MOVL C00616 V=800.0 PL=0
MOVL C00617 V=800.0 PL=0
MOVL C00618 V=800.0 PL=0
MOVL C00619 V=800.0 PL=0
MOVL C00620 V=800.0 PL=0
MOVL C00621 V=800.0 PL=0
MOVL C00622 V=800.0 PL=0
MOVL C00623 V=800.0 PL=0
MOVL C00624 V=800.0 PL=0
MOVL C00625 V=800.0 PL=0
MOVL C00626 V=800.0 PL=0
MOVL C00627 V=800.0 PL=0
MOVL C00628 V=800.0 PL=0
MOVL C00629 V=800.0 PL=0
MOVL C00630 V=800.0 PL=0
MOVL C00631 V=800.0 PL=0
MOVL C00632 V=800.0 PL=0
MOVL C00633 V=800.0 PL=0
MOVL C00634 V=800.0 PL=0
MOVL C00635 V=800.0 PL=0
MOVL C00636 V=800.0 PL=0
MOVL C00637 V=800.0 PL=0
MOVL C00638 V=800.0 PL=0
MOVL C00639 V=800.0 PL=0
MOVL C00640 V=800.0 PL=0
MOVL C00641 V=800.0 PL=0
MOVL C00642 V=800.0 PL=0
MOVL C00643 V=800.0 PL=0
MOVL C00644 V=800.0 PL=0
MOVL C00645 V=800.0 PL=0
MOVL C00646 V=800.0 PL=0
MOVL C00647 V=800.0 PL=0
MOVL C00648 V=800.0 PL=0
MOVL C00649 V=800.0 PL=0
MOVL C00650 V=800.0 PL=0
MOVL C00651 V=800.0 PL=0
MOVL C00652 V=800.0 PL=0
MOVL C00653 V=800.0 PL=0
MOVL C00654 V=800.0 PL=0
MOVL C00655 V=800.0 PL=0
MOVL C00656 V=800.0 PL=0
MOVL C00657 V=800.0 PL=0
MOVL C00658 V=800.0 PL=0
MOVL C00659 V=800.0 PL=0
MOVL C00660 V=800.0 PL=0
MOVL C00661 V=800.0 PL=0
MOVL C00662 V=800.0 PL=0
MOVL C00663 V=800.0 PL=0
MOVL C00664 V=800.0 PL=0
MOVL C00665 V=800.0 PL=0
MOVL C00666 V=800.0 PL=0
MOVL C00667 V=800.0 PL=0
MOVL C00668 V=800.0 PL=0
MOVL C00669 V=800.0 PL=0
MOVL C00670 V=800.0 PL=0
MOVL C00671 V=800.0 PL=0
MOVL C00672 V=800.0 PL=0
MOVL C00673 V=800.0 PL=0
MOVL C00674 V=800.0 PL=0
MOVL C00675 V=800.0 PL=0
MOVL C00676 V=800.0 PL=0
MOVL C00677 V=800.0 PL=0
MOVL C00678 V=800.0 PL=0
MOVL C00679 V=800.0 PL=0
MOVL C00680 V=800.0 PL=0
MOVL C00681 V=800.0 PL=0
MOVL C00682 V=800.0 PL=0
MOVL C00683 V=800.0 PL=0
MOVL C00684 V=800.0 PL=0
MOVL C00685 V=800.0 PL=0
MOVL C00686 V=800.0 PL=0
MOVL C00687 V=800.0 PL=0
MOVL C00688 V=800.0 PL=0
MOVL C00689 V=800.0 PL=0
MOVL C00690 V=800.0 PL=0
MOVL C00691 V=800.0 PL=0
MOVL C00692 V=800.0 PL=0
MOVL C00693 V=800.0 PL=0
MOVL C00694 V=800.0 PL=0
MOVL C00695 V=800.0 PL=0
MOVL C00696 V=800.0 PL=0
MOVL C00697 V=800.0 PL=0
MOVL C00698 V=800.0 PL=0
MOVL C00699 V=800.0 PL=0
MOVL C00700 V=800.0 PL=0
MOVL C00701 V=800.0 PL=0
MOVL C00702 V=800.0 PL=0
MOVL C00703 V=800.0 PL=0
MOVL C00704 V=800.0 PL=0
MOVL C00705 V=800.0 PL=0
MOVL C00706 V=800.0 PL=0
MOVL C00707 V=800.0 PL=0
MOVL C00708 V=800.0 PL=0
MOVL C00709 V=800.0 PL=0
MOVL C00710 V=800.0 PL=0
MOVL C00711 V=800.0 PL=0
MOVL C00712 V=800.0 PL=0
MOVL C00713 V=800.0 PL=0
MOVL C00714 V=800.0 PL=0
MOVL C00715 V=800.0 PL=0
MOVL C00716 V=800.0 PL=0
MOVL C00717 V=800.0 PL=0
MOVL C00718 V=800.0 PL=0
MOVL C00719 V=800.0 PL=0
MOVL C00720 V=800.0 PL=0
MOVL C00721 V=800.0 PL=0
MOVL C00722 V=800.0 PL=0
MOVL C00723 V=800.0 PL=0
MOVL C00724 V=800.0 PL=0
MOVL C00725 V=800.0 PL=0
MOVL C00726 V=800.0 PL=0
MOVL C00727 V=800.0 PL=0
MOVL C00728 V=800.0 PL=0
MOVL C00729 V=800.0 PL=0
MOVL C00730 V=800.0 PL=0
MOVL C00731 V=800.0 PL=0
MOVL C00732 V=800.0 PL=0
MOVL C00733 V=800.0 PL=0
MOVL C00734 V=800.0 PL=0
MOVL C00735 V=800.0 PL=0
MOVL C00736 V=800.0 PL=0
MOVL C00737 V=800.0 PL=0
MOVL C00738 V=800.0 PL=0
MOVL C00739 V=800.0 PL=0
MOVL C00740 V=800.0 PL=0
MOVL C00741 V=800.0 PL=0
MOVL C00742 V=800.0 PL=0
MOVL C00743 V=800.0 PL=0
MOVL C00744 V=800.0 PL=0
MOVL C00745 V=800.0 PL=0
MOVL C00746 V=800.0 PL=0
MOVL C00747 V=800.0 PL=0
MOVL C00748 V=800.0 PL=0
MOVL C00749 V=800.0 PL=0
MOVL C00750 V=800.0 PL=0
MOVL C00751 V=800.0 PL=0
MOVL C00752 V=800.0 PL=0
MOVL C00753 V=800.0 PL=0
MOVL C00754 V=800.0 PL=0
MOVL C00755 V=800.0 PL=0
MOVL C00756 V=800.0 PL=0
MOVL C00757 V=800.0 PL=0
MOVL C00758 V=800.0 PL=0
MOVL C00759 V=800.0 PL=0
MOVL C00760 V=800.0 PL=0
MOVL C00761 V=800.0 PL=0
MOVL C00762 V=800.0 PL=0
MOVL C00763 V=800.0 PL=0
MOVL C00764 V=800.0 PL=0
MOVL C00765 V=800.0 PL=0
MOVL C00766 V=800.0 PL=0
MOVL C00767 V=800.0 PL=0
MOVL C00768 V=800.0 PL=0
MOVL C00769 V=800.0 PL=0
MOVL C00770 V=800.0 PL=0
MOVL C00771 V=800.0 PL=0
MOVL C00772 V=800.0 PL=0
MOVL C00773 V=800.0 PL=0
MOVL C00774 V=800.0 PL=0
MOVL C00775 V=800.0 PL=0
MOVL C00776 V=800.0 PL=0
MOVL C00777 V=800.0 PL=0
MOVL C00778 V=800.0 PL=0
MOVL C00779 V=800.0 PL=0
MOVL C00780 V=800.0 PL=0
MOVL C00781 V=800.0 PL=0
MOVL C00782 V=800.0 PL=0
MOVL C00783 V=800.0 PL=0
MOVL C00784 V=800.0 PL=0
MOVL C00785 V=800.0 PL=0
MOVL C00786 V=800.0 PL=0
MOVL C00787 V=800.0 PL=0
MOVL C00788 V=800.0 PL=0
MOVL C00789 V=800.0 PL=0
MOVL C00790 V=800.0 PL=0
MOVL C00791 V=800.0 PL=0
MOVL C00792 V=800.0 PL=0
MOVL C00793 V=800.0 PL=0
MOVL C00794 V=800.0 PL=0
MOVL C00795 V=800.0 PL=0
MOVL C00796 V=800.0 PL=0
MOVL C00797 V=800.0 PL=0
MOVL C00798 V=800.0 PL=0
MOVL C00799 V=800.0 PL=0
MOVL C00800 V=800.0 PL=0
MOVL C00801 V=800.0 PL=0
MOVL C00802 V=800.0 PL=0
MOVL C00803 V=800.0 PL=0
MOVL C00804 V=800.0 PL=0
MOVL C00805 V=800.0 PL=0
MOVL C00806 V=800.0 PL=0
MOVL C00807 V=800.0 PL=0
MOVL C00808 V=800.0 PL=0
MOVL C00809 V=800.0 PL=0
MOVL C00810 V=800.0 PL=0
MOVL C00811 V=800.0 PL=0
MOVL C00812 V=800.0 PL=0
MOVL C00813 V=800.0 PL=0
MOVL C00814 V=800.0 PL=0
MOVL C00815 V=800.0 PL=0
MOVL C00816 V=800.0 PL=0
MOVL C00817 V=800.0 PL=0
MOVL C00818 V=800.0 PL=0
MOVL C00819 V=800.0 PL=0
MOVL C00820 V=800.0 PL=0
MOVL C00821 V=800.0 PL=0
MOVL C00822 V=800.0 PL=0
MOVL C00823 V=800.0 PL=0
MOVL C00824 V=800.0 PL=0
MOVL C00825 V=800.0 PL=0
MOVL C00826 V=800.0 PL=0
MOVL C00827 V=800.0 PL=0
MOVL C00828 V=800.0 PL=0
MOVL C00829 V=800.0 PL=0
MOVL C00830 V=800.0 PL=0
MOVL C00831 V=800.0 PL=0
MOVL C00832 V=800.0 PL=0
MOVL C00833 V=800.0 PL=0
MOVL C00834 V=800.0 PL=0
MOVL C00835 V=800.0 PL=0
MOVL C00836 V=800.0 PL=0
MOVL C00837 V=800.0 PL=0
MOVL C00838 V=800.0 PL=0
MOVL C00839 V=800.0 PL=0
MOVL C00840 V=800.0 PL=0
MOVL C00841 V=800.0 PL=0
MOVL C00842 V=800.0 PL=0
MOVL C00843 V=800.0 PL=0
MOVL C00844 V=800.0 PL=0
MOVL C00845 V=800.0 PL=0
MOVL C00846 V=800.0 PL=0
MOVL C00847 V=800.0 PL=0
MOVL C00848 V=800.0 PL=0
MOVL C00849 V=800.0 PL=0
MOVL C00850 V=800.0 PL=0
MOVL C00851 V=800.0 PL=0
MOVL C00852 V=800.0 PL=0
MOVL C00853 V=800.0 PL=0
MOVL C00854 V=800.0 PL=0
MOVL C00855 V=800.0 PL=0
MOVL C00856 V=800.0 PL=0
MOVL C00857 V=800.0 PL=0
MOVL C00858 V=800.0 PL=0
MOVL C00859 V=800.0 PL=0
MOVL C00860 V=800.0 PL=0
MOVL C00861 V=800.0 PL=0
MOVL C00862 V=800.0 PL=0
MOVL C00863 V=800.0 PL=0
MOVL C00864 V=800.0 PL=0
MOVL C00865 V=800.0 PL=0
MOVL C00866 V=800.0 PL=0
MOVL C00867 V=800.0 PL=0
MOVL C00868 V=800.0 PL=0
MOVL C00869 V=800.0 PL=0
MOVL C00870 V=800.0 PL=0
MOVL C00871 V=800.0 PL=0
MOVL C00872 V=800.0 PL=0
MOVL C00873 V=800.0 PL=0
MOVL C00874 V=800.0 PL=0
MOVL C00875 V=800.0 PL=0
MOVL C00876 V=800.0 PL=0
MOVL C00877 V=800.0 PL=0
MOVL C00878 V=800.0 PL=0
MOVL C00879 V=800.0 PL=0
MOVL C00880 V=800.0 PL=0
MOVL C00881 V=800.0 PL=0
MOVL C00882 V=800.0 PL=0
MOVL C00883 V=800.0 PL=0
MOVL C00884 V=800.0 PL=0
MOVL C00885 V=800.0 PL=0
MOVL C00886 V=800.0 PL=0
MOVL C00887 V=800.0 PL=0
MOVL C00888 V=800.0 PL=0
MOVL C00889 V=800.0 PL=0
MOVL C00890 V=800.0 PL=0
MOVL C00891 V=800.0 PL=0
MOVL C00892 V=800.0 PL=0
MOVL C00893 V=800.0 PL=0
MOVL C00894 V=800.0 PL=0
MOVL C00895 V=800.0 PL=0
MOVL C00896 V=800.0 PL=0
MOVL C00897 V=800.0 PL=0
MOVL C00898 V=800.0 PL=0
MOVL C00899 V=800.0 PL=0
MOVL C00900 V=800.0 PL=0
MOVL C00901 V=800.0 PL=0
MOVL C00902 V=800.0 PL=0
MOVL C00903 V=800.0 PL=0
MOVL C00904 V=800.0 PL=0
MOVL C00905 V=800.0 PL=0
MOVL C00906 V=800.0 PL=0
MOVL C00907 V=800.0 PL=0
MOVL C00908 V=800.0 PL=0
MOVL C00909 V=800.0 PL=0
MOVL C00910 V=800.0 PL=0
MOVL C00911 V=800.0 PL=0
MOVL C00912 V=800.0 PL=0
MOVL C00913 V=800.0 PL=0
MOVL C00914 V=800.0 PL=0
MOVL C00915 V=800.0 PL=0
MOVL C00916 V=800.0 PL=0
MOVL C00917 V=800.0 PL=0
MOVL C00918 V=800.0 PL=0
MOVL C00919 V=800.0 PL=0
MOVL C00920 V=800.0 PL=0
MOVL C00921 V=800.0 PL=0
MOVL C00922 V=800.0 PL=0
MOVL C00923 V=800.0 PL=0
MOVL C00924 V=800.0 PL=0
MOVL C00925 V=800.0 PL=0
MOVL C00926 V=800.0 PL=0
MOVL C00927 V=800.0 PL=0
MOVL C00928 V=800.0 PL=0
MOVL C00929 V=800.0 PL=0
MOVL C00930 V=800.0 PL=0
MOVL C00931 V=800.0 PL=0
MOVL C00932 V=800.0 PL=0
MOVL C00933 V=800.0 PL=0
MOVL C00934 V=800.0 PL=0
MOVL C00935 V=800.0 PL=0
MOVL C00936 V=800.0 PL=0
MOVL C00937 V=800.0 PL=0
MOVL C00938 V=800.0 PL=0
MOVL C00939 V=800.0 PL=0
MOVL C00940 V=800.0 PL=0
MOVL C00941 V=800.0 PL=0
MOVL C00942 V=800.0 PL=0
MOVL C00943 V=800.0 PL=0
MOVL C00944 V=800.0 PL=0
MOVL C00945 V=800.0 PL=0
MOVL C00946 V=800.0 PL=0
MOVL C00947 V=800.0 PL=0
MOVL C00948 V=800.0 PL=0
MOVL C00949 V=800.0 PL=0
MOVL C00950 V=800.0 PL=0
MOVL C00951 V=800.0 PL=0
MOVL C00952 V=800.0 PL=0
MOVL C00953 V=800.0 PL=0
MOVL C00954 V=800.0 PL=0
MOVL C00955 V=800.0 PL=0
MOVL C00956 V=800.0 PL=0
MOVL C00957 V=800.0 PL=0
MOVL C00958 V=800.0 PL=0
MOVL C00959 V=800.0 PL=0
MOVL C00960 V=800.0 PL=0
MOVL C00961 V=800.0 PL=0
MOVL C00962 V=800.0 PL=0
MOVL C00963 V=800.0 PL=0
MOVL C00964 V=800.0 PL=0
MOVL C00965 V=800.0 PL=0
MOVL C00966 V=800.0 PL=0
MOVL C00967 V=800.0 PL=0
MOVL C00968 V=800.0 PL=0
MOVL C00969 V=800.0 PL=0
MOVL C00970 V=800.0 PL=0
MOVL C00971 V=800.0 PL=0
MOVL C00972 V=800.0 PL=0
MOVL C00973 V=800.0 PL=0
MOVL C00974 V=800.0 PL=0
MOVL C00975 V=800.0 PL=0
MOVL C00976 V=800.0 PL=0
MOVL C00977 V=800.0 PL=0
MOVL C00978 V=800.0 PL=0
MOVL C00979 V=800.0 PL=0
MOVL C00980 V=800.0 PL=0
MOVL C00981 V=800.0 PL=0
MOVL C00982 V=800.0 PL=0
MOVL C00983 V=800.0 PL=0
MOVL C00984 V=800.0 PL=0
MOVL C00985 V=800.0 PL=0
MOVL C00986 V=800.0 PL=0
MOVL C00987 V=800.0 PL=0
MOVL C00988 V=800.0 PL=0
MOVL C00989 V=800.0 PL=0
MOVL C00990 V=800.0 PL=0
MOVL C00991 V=800.0 PL=0
MOVL C00992 V=800.0 PL=0
MOVL C00993 V=800.0 PL=0
MOVL C00994 V=800.0 PL=0
MOVL C00995 V=800.0 PL=0
MOVL C00996 V=800.0 PL=0
MOVL C00997 V=800.0 PL=0
MOVL C00998 V=800.0 PL=0
MOVL C00999 V=800.0 PL=0
MOVL C01000 V=800.0 PL=0
MOVL C01001 V=800.0 PL=0
MOVL C01002 V=800.0 PL=0
MOVL C01003 V=800.0 PL=0
MOVL C01004 V=800.0 PL=0
MOVL C01005 V=800.0 PL=0
MOVL C01006 V=800.0 PL=0
MOVL C01007 V=800.0 PL=0
MOVL C01008 V=800.0 PL=0
MOVL C01009 V=800.0 PL=0
MOVL C01010 V=800.0 PL=0
MOVL C01011 V=800.0 PL=0
MOVL C01012 V=800.0 PL=0
MOVL C01013 V=800.0 PL=0
MOVL C01014 V=800.0 PL=0
MOVL C01015 V=800.0 PL=0
MOVL C01016 V=800.0 PL=0
MOVL C01017 V=800.0 PL=0
MOVL C01018 V=800.0 PL=0
MOVL C01019 V=800.0 PL=0
MOVL C01020 V=800.0 PL=0
MOVL C01021 V=800.0 PL=0
MOVL C01022 V=800.0 PL=0
MOVL C01023 V=800.0 PL=0
MOVL C01024 V=800.0 PL=0
MOVL C01025 V=800.0 PL=0
MOVL C01026 V=800.0 PL=0
MOVL C01027 V=800.0 PL=0
MOVL C01028 V=800.0 PL=0
MOVL C01029 V=800.0 PL=0
MOVL C01030 V=800.0 PL=0
MOVL C01031 V=800.0 PL=0
MOVL C01032 V=800.0 PL=0
MOVL C01033 V=800.0 PL=0
MOVL C01034 V=800.0 PL=0
MOVL C01035 V=800.0 PL=0
MOVL C01036 V=800.0 PL=0
MOVL C01037 V=800.0 PL=0
MOVL C01038 V=800.0 PL=0
MOVL C01039 V=800.0 PL=0
MOVL C01040 V=800.0 PL=0
MOVL C01041 V=800.0 PL=0
MOVL C01042 V=800.0 PL=0
MOVL C01043 V=800.0 PL=0
MOVL C01044 V=800.0 PL=0
MOVL C01045 V=800.0 PL=0
MOVL C01046 V=800.0 PL=0
MOVL C01047 V=800.0 PL=0
MOVL C01048 V=800.0 PL=0
MOVL C01049 V=800.0 PL=0
MOVL C01050 V=800.0 PL=0
MOVL C01051 V=800.0 PL=0
MOVL C01052 V=800.0 PL=0
MOVL C01053 V=800.0 PL=0
MOVL C01054 V=800.0 PL=0
MOVL C01055 V=800.0 PL=0
MOVL C01056 V=800.0 PL=0
MOVL C01057 V=800.0 PL=0
MOVL C01058 V=800.0 PL=0
MOVL C01059 V=800.0 PL=0
MOVL C01060 V=800.0 PL=0
MOVL C01061 V=800.0 PL=0
MOVL C01062 V=800.0 PL=0
MOVL C01063 V=800.0 PL=0
MOVL C01064 V=800.0 PL=0
MOVL C01065 V=800.0 PL=0
MOVL C01066 V=800.0 PL=0
MOVL C01067 V=800.0 PL=0
MOVL C01068 V=800.0 PL=0
MOVL C01069 V=800.0 PL=0
MOVL C01070 V=800.0 PL=0
MOVL C01071 V=800.0 PL=0
MOVL C01072 V=800.0 PL=0
MOVL C01073 V=800.0 PL=0
MOVL C01074 V=800.0 PL=0
MOVL C01075 V=800.0 PL=0
MOVL C01076 V=800.0 PL=0
MOVL C01077 V=800.0 PL=0
MOVL C01078 V=800.0 PL=0
MOVL C01079 V=800.0 PL=0
MOVL C01080 V=800.0 PL=0
MOVL C01081 V=800.0 PL=0
MOVL C01082 V=800.0 PL=0
MOVL C01083 V=800.0 PL=0
MOVL C01084 V=800.0 PL=0
MOVL C01085 V=800.0 PL=0
MOVL C01086 V=800.0 PL=0
MOVL C01087 V=800.0 PL=0
MOVL C01088 V=800.0 PL=0
MOVL C01089 V=800.0 PL=0
MOVL C01090 V=800.0 PL=0
MOVL C01091 V=800.0 PL=0
MOVL C01092 V=800.0 PL=0
MOVL C01093 V=800.0 PL=0
MOVL C01094 V=800.0 PL=0
MOVL C01095 V=800.0 PL=0
MOVL C01096 V=800.0 PL=0
MOVL C01097 V=800.0 PL=0
MOVL C01098 V=800.0 PL=0
MOVL C01099 V=800.0 PL=0
MOVL C01100 V=800.0 PL=0
MOVL C01101 V=800.0 PL=0
MOVL C01102 V=800.0 PL=0
MOVL C01103 V=800.0 PL=0
MOVL C01104 V=800.0 PL=0
MOVL C01105 V=800.0 PL=0
MOVL C01106 V=800.0 PL=0
MOVL C01107 V=800.0 PL=0
MOVL C01108 V=800.0 PL=0
MOVL C01109 V=800.0 PL=0
MOVL C01110 V=800.0 PL=0
MOVL C01111 V=800.0 PL=0
MOVL C01112 V=800.0 PL=0
MOVL C01113 V=800.0 PL=0
MOVL C01114 V=800.0 PL=0
MOVL C01115 V=800.0 PL=0
MOVL C01116 V=800.0 PL=0
MOVL C01117 V=800.0 PL=0
MOVL C01118 V=800.0 PL=0
MOVL C01119 V=800.0 PL=0
MOVL C01120 V=800.0 PL=0
MOVL C01121 V=800.0 PL=0
MOVL C01122 V=800.0 PL=0
MOVL C01123 V=800.0 PL=0
MOVL C01124 V=800.0 PL=0
MOVL C01125 V=800.0 PL=0
MOVL C01126 V=800.0 PL=0
MOVL C01127 V=800.0 PL=0
MOVL C01128 V=800.0 PL=0
MOVL C01129 V=800.0 PL=0
MOVL C01130 V=800.0 PL=0
MOVL C01131 V=800.0 PL=0
MOVL C01132 V=800.0 PL=0
MOVL C01133 V=800.0 PL=0
MOVL C01134 V=800.0 PL=0
MOVL C01135 V=800.0 PL=0
MOVL C01136 V=800.0 PL=0
MOVL C01137 V=800.0 PL=0
MOVL C01138 V=800.0 PL=0
MOVL C01139 V=800.0 PL=0
MOVL C01140 V=800.0 PL=0
MOVL C01141 V=800.0 PL=0
MOVL C01142 V=800.0 PL=0
MOVL C01143 V=800.0 PL=0
MOVL C01144 V=800.0 PL=0
MOVL C01145 V=800.0 PL=0
MOVL C01146 V=800.0 PL=0
MOVL C01147 V=800.0 PL=0
MOVL C01148 V=800.0 PL=0
MOVL C01149 V=800.0 PL=0
MOVL C01150 V=800.0 PL=0
MOVL C01151 V=800.0 PL=0
MOVL C01152 V=800.0 PL=0
MOVL C01153 V=800.0 PL=0
MOVL C01154 V=800.0 PL=0
MOVL C01155 V=800.0 PL=0
MOVL C01156 V=800.0 PL=0
MOVL C01157 V=800.0 PL=0
MOVL C01158 V=800.0 PL=0
MOVL C01159 V=800.0 PL=0
MOVL C01160 V=800.0 PL=0
MOVL C01161 V=800.0 PL=0
MOVL C01162 V=800.0 PL=0
MOVL C01163 V=800.0 PL=0
MOVL C01164 V=800.0 PL=0
MOVL C01165 V=800.0 PL=0
MOVL C01166 V=800.0 PL=0
MOVL C01167 V=800.0 PL=0
MOVL C01168 V=800.0 PL=0
MOVL C01169 V=800.0 PL=0
MOVL C01170 V=800.0 PL=0
MOVL C01171 V=800.0 PL=0
MOVL C01172 V=800.0 PL=0
MOVL C01173 V=800.0 PL=0
MOVL C01174 V=800.0 PL=0
MOVL C01175 V=800.0 PL=0
MOVL C01176 V=800.0 PL=0
MOVL C01177 V=800.0 PL=0
MOVL C01178 V=800.0 PL=0
MOVL C01179 V=800.0 PL=0
MOVL C01180 V=800.0 PL=0
MOVL C01181 V=800.0 PL=0
MOVL C01182 V=800.0 PL=0
MOVL C01183 V=800.0 PL=0
MOVL C01184 V=800.0 PL=0
MOVL C01185 V=800.0 PL=0
MOVL C01186 V=800.0 PL=0
MOVL C01187 V=800.0 PL=0
MOVL C01188 V=800.0 PL=0
MOVL C01189 V=800.0 PL=0
MOVL C01190 V=800.0 PL=0
MOVL C01191 V=800.0 PL=0
MOVL C01192 V=800.0 PL=0
MOVL C01193 V=800.0 PL=0
MOVL C01194 V=800.0 PL=0
MOVL C01195 V=800.0 PL=0
MOVL C01196 V=800.0 PL=0
MOVL C01197 V=800.0 PL=0
MOVL C01198 V=800.0 PL=0
MOVL C01199 V=800.0 PL=0
MOVL C01200 V=800.0 PL=0
MOVL C01201 V=800.0 PL=0
MOVL C01202 V=800.0 PL=0
MOVL C01203 V=800.0 PL=0
MOVL C01204 V=800.0 PL=0
MOVL C01205 V=800.0 PL=0
MOVL C01206 V=800.0 PL=0
MOVL C01207 V=800.0 PL=0
MOVL C01208 V=800.0 PL=0
MOVL C01209 V=800.0 PL=0
MOVL C01210 V=800.0 PL=0
MOVL C01211 V=800.0 PL=0
MOVL C01212 V=800.0 PL=0
MOVL C01213 V=800.0 PL=0
MOVL C01214 V=800.0 PL=0
MOVL C01215 V=800.0 PL=0
MOVL C01216 V=800.0 PL=0
MOVL C01217 V=800.0 PL=0
MOVL C01218 V=800.0 PL=0
MOVL C01219 V=800.0 PL=0
MOVL C01220 V=800.0 PL=0
MOVL C01221 V=800.0 PL=0
MOVL C01222 V=800.0 PL=0
MOVL C01223 V=800.0 PL=0
MOVL C01224 V=800.0 PL=0
MOVL C01225 V=800.0 PL=0
MOVL C01226 V=800.0 PL=0
MOVL C01227 V=800.0 PL=0
MOVL C01228 V=800.0 PL=0
MOVL C01229 V=800.0 PL=0
MOVL C01230 V=800.0 PL=0
MOVL C01231 V=800.0 PL=0
MOVL C01232 V=800.0 PL=0
MOVL C01233 V=800.0 PL=0
MOVL C01234 V=800.0 PL=0
MOVL C01235 V=800.0 PL=0
MOVL C01236 V=800.0 PL=0
MOVL C01237 V=800.0 PL=0
MOVL C01238 V=800.0 PL=0
MOVL C01239 V=800.0 PL=0
MOVL C01240 V=800.0 PL=0
MOVL C01241 V=800.0 PL=0
MOVL C01242 V=800.0 PL=0
MOVL C01243 V=800.0 PL=0
MOVL C01244 V=800.0 PL=0
MOVL C01245 V=800.0 PL=0
MOVL C01246 V=800.0 PL=0
MOVL C01247 V=800.0 PL=0
MOVL C01248 V=800.0 PL=0
MOVL C01249 V=800.0 PL=0
MOVL C01250 V=800.0 PL=0
MOVL C01251 V=800.0 PL=0
MOVL C01252 V=800.0 PL=0
MOVL C01253 V=800.0 PL=0
MOVL C01254 V=800.0 PL=0
MOVL C01255 V=800.0 PL=0
MOVL C01256 V=800.0 PL=0
MOVL C01257 V=800.0 PL=0
MOVL C01258 V=800.0 PL=0
MOVL C01259 V=800.0 PL=0
MOVL C01260 V=800.0 PL=0
MOVL C01261 V=800.0 PL=0
MOVL C01262 V=800.0 PL=0
MOVL C01263 V=800.0 PL=0
MOVL C01264 V=800.0 PL=0
MOVL C01265 V=800.0 PL=0
MOVL C01266 V=800.0 PL=0
MOVL C01267 V=800.0 PL=0
MOVL C01268 V=800.0 PL=0
MOVL C01269 V=800.0 PL=0
MOVL C01270 V=800.0 PL=0
MOVL C01271 V=800.0 PL=0
MOVL C01272 V=800.0 PL=0
MOVL C01273 V=800.0 PL=0
MOVL C01274 V=800.0 PL=0
MOVL C01275 V=800.0 PL=0
MOVL C01276 V=800.0 PL=0
MOVL C01277 V=800.0 PL=0
MOVL C01278 V=800.0 PL=0
MOVL C01279 V=800.0 PL=0
MOVL C01280 V=800.0 PL=0
MOVL C01281 V=800.0 PL=0
MOVL C01282 V=800.0 PL=0
MOVL C01283 V=800.0 PL=0
MOVL C01284 V=800.0 PL=0
MOVL C01285 V=800.0 PL=0
MOVL C01286 V=800.0 PL=0
MOVL C01287 V=800.0 PL=0
MOVL C01288 V=800.0 PL=0
MOVL C01289 V=800.0 PL=0
MOVL C01290 V=800.0 PL=0
MOVL C01291 V=800.0 PL=0
MOVL C01292 V=800.0 PL=0
MOVL C01293 V=800.0 PL=0
MOVL C01294 V=800.0 PL=0
MOVL C01295 V=800.0 PL=0
MOVL C01296 V=800.0 PL=0
MOVL C01297 V=800.0 PL=0
MOVL C01298 V=800.0 PL=0
MOVL C01299 V=800.0 PL=0
MOVL C01300 V=800.0 PL=0
MOVL C01301 V=800.0 PL=0
MOVL C01302 V=800.0 PL=0
MOVL C01303 V=800.0 PL=0
MOVL C01304 V=800.0 PL=0
MOVL C01305 V=800.0 PL=0
MOVL C01306 V=800.0 PL=0
MOVL C01307 V=800.0 PL=0
MOVL C01308 V=800.0 PL=0
MOVL C01309 V=800.0 PL=0
MOVL C01310 V=800.0 PL=0
MOVL C01311 V=800.0 PL=0
MOVL C01312 V=800.0 PL=0
MOVL C01313 V=800.0 PL=0
MOVL C01314 V=800.0 PL=0
MOVL C01315 V=800.0 PL=0
MOVL C01316 V=800.0 PL=0
MOVL C01317 V=800.0 PL=0
MOVL C01318 V=800.0 PL=0
MOVL C01319 V=800.0 PL=0
MOVL C01320 V=800.0 PL=0
MOVL C01321 V=800.0 PL=0
MOVL C01322 V=800.0 PL=0
MOVL C01323 V=800.0 PL=0
MOVL C01324 V=800.0 PL=0
MOVL C01325 V=800.0 PL=0
MOVL C01326 V=800.0 PL=0
MOVL C01327 V=800.0 PL=0
MOVL C01328 V=800.0 PL=0
MOVL C01329 V=800.0 PL=0
MOVL C01330 V=800.0 PL=0
MOVL C01331 V=800.0 PL=0
MOVL C01332 V=800.0 PL=0
MOVL C01333 V=800.0 PL=0
MOVL C01334 V=800.0 PL=0
MOVL C01335 V=800.0 PL=0
MOVL C01336 V=800.0 PL=0
MOVL C01337 V=800.0 PL=0
MOVL C01338 V=800.0 PL=0
MOVL C01339 V=800.0 PL=0
MOVL C01340 V=800.0 PL=0
MOVL C01341 V=800.0 PL=0
MOVL C01342 V=800.0 PL=0
MOVL C01343 V=800.0 PL=0
MOVL C01344 V=800.0 PL=0
MOVL C01345 V=800.0 PL=0
MOVL C01346 V=800.0 PL=0
MOVL C01347 V=800.0 PL=0
MOVL C01348 V=800.0 PL=0
MOVL C01349 V=800.0 PL=0
MOVL C01350 V=800.0 PL=0
MOVL C01351 V=800.0 PL=0
MOVL C01352 V=800.0 PL=0
MOVL C01353 V=800.0 PL=0
MOVL C01354 V=800.0 PL=0
MOVL C01355 V=800.0 PL=0
MOVL C01356 V=800.0 PL=0
MOVL C01357 V=800.0 PL=0
MOVL C01358 V=800.0 PL=0
MOVL C01359 V=800.0 PL=0
MOVL C01360 V=800.0 PL=0
MOVL C01361 V=800.0 PL=0
MOVL C01362 V=800.0 PL=0
MOVL C01363 V=800.0 PL=0
MOVL C01364 V=800.0 PL=0
MOVL C01365 V=800.0 PL=0
MOVL C01366 V=800.0 PL=0
MOVL C01367 V=800.0 PL=0
MOVL C01368 V=800.0 PL=0
MOVL C01369 V=800.0 PL=0
MOVL C01370 V=800.0 PL=0
MOVL C01371 V=800.0 PL=0
MOVL C01372 V=800.0 PL=0
MOVL C01373 V=800.0 PL=0
MOVL C01374 V=800.0 PL=0
MOVL C01375 V=800.0 PL=0
MOVL C01376 V=800.0 PL=0
MOVL C01377 V=800.0 PL=0
MOVL C01378 V=800.0 PL=0
MOVL C01379 V=800.0 PL=0
MOVL C01380 V=800.0 PL=0
MOVL C01381 V=800.0 PL=0
MOVL C01382 V=800.0 PL=0
MOVL C01383 V=800.0 PL=0
MOVL C01384 V=800.0 PL=0
MOVL C01385 V=800.0 PL=0
MOVL C01386 V=800.0 PL=0
MOVL C01387 V=800.0 PL=0
MOVL C01388 V=800.0 PL=0
MOVL C01389 V=800.0 PL=0
MOVL C01390 V=800.0 PL=0
MOVL C01391 V=800.0 PL=0
MOVL C01392 V=800.0 PL=0
MOVL C01393 V=800.0 PL=0
MOVL C01394 V=800.0 PL=0
MOVL C01395 V=800.0 PL=0
MOVL C01396 V=800.0 PL=0
MOVL C01397 V=800.0 PL=0
MOVL C01398 V=800.0 PL=0
MOVL C01399 V=800.0 PL=0
MOVL C01400 V=800.0 PL=0
MOVL C01401 V=800.0 PL=0
MOVL C01402 V=800.0 PL=0
MOVL C01403 V=800.0 PL=0
MOVL C01404 V=800.0 PL=0
MOVL C01405 V=800.0 PL=0
MOVL C01406 V=800.0 PL=0
MOVL C01407 V=800.0 PL=0
MOVL C01408 V=800.0 PL=0
MOVL C01409 V=800.0 PL=0
MOVL C01410 V=800.0 PL=0
MOVL C01411 V=800.0 PL=0
MOVL C01412 V=800.0 PL=0
MOVL C01413 V=800.0 PL=0
MOVL C01414 V=800.0 PL=0
MOVL C01415 V=800.0 PL=0
MOVL C01416 V=800.0 PL=0
MOVL C01417 V=800.0 PL=0
MOVL C01418 V=800.0 PL=0
MOVL C01419 V=800.0 PL=0
MOVL C01420 V=800.0 PL=0
MOVL C01421 V=800.0 PL=0
MOVL C01422 V=800.0 PL=0
MOVL C01423 V=800.0 PL=0
MOVL C01424 V=800.0 PL=0
MOVL C01425 V=800.0 PL=0
MOVL C01426 V=800.0 PL=0
MOVL C01427 V=800.0 PL=0
MOVL C01428 V=800.0 PL=0
MOVL C01429 V=800.0 PL=0
MOVL C01430 V=800.0 PL=0
MOVL C01431 V=800.0 PL=0
MOVL C01432 V=800.0 PL=0
MOVL C01433 V=800.0 PL=0
MOVL C01434 V=800.0 PL=0
MOVL C01435 V=800.0 PL=0
MOVL C01436 V=800.0 PL=0
MOVL C01437 V=800.0 PL=0
MOVL C01438 V=800.0 PL=0
MOVL C01439 V=800.0 PL=0
MOVL C01440 V=800.0 PL=0
MOVL C01441 V=800.0 PL=0
MOVL C01442 V=800.0 PL=0
MOVL C01443 V=800.0 PL=0
MOVL C01444 V=800.0 PL=0
MOVL C01445 V=800.0 PL=0
MOVL C01446 V=800.0 PL=0
MOVL C01447 V=800.0 PL=0
MOVL C01448 V=800.0 PL=0
MOVL C01449 V=800.0 PL=0
MOVL C01450 V=800.0 PL=0
MOVL C01451 V=800.0 PL=0
MOVL C01452 V=800.0 PL=0
MOVL C01453 V=800.0 PL=0
MOVL C01454 V=800.0 PL=0
MOVL C01455 V=800.0 PL=0
MOVL C01456 V=800.0 PL=0
MOVL C01457 V=800.0 PL=0
MOVL C01458 V=800.0 PL=0
MOVL C01459 V=800.0 PL=0
MOVL C01460 V=800.0 PL=0
MOVL C01461 V=800.0 PL=0
MOVL C01462 V=800.0 PL=0
MOVL C01463 V=800.0 PL=0
MOVL C01464 V=800.0 PL=0
MOVL C01465 V=800.0 PL=0
MOVL C01466 V=800.0 PL=0
MOVL C01467 V=800.0 PL=0
MOVL C01468 V=800.0 PL=0
MOVL C01469 V=800.0 PL=0
MOVL C01470 V=800.0 PL=0
MOVL C01471 V=800.0 PL=0
MOVL C01472 V=800.0 PL=0
MOVL C01473 V=800.0 PL=0
MOVL C01474 V=800.0 PL=0
MOVL C01475 V=800.0 PL=0
MOVL C01476 V=800.0 PL=0
MOVL C01477 V=800.0 PL=0
MOVL C01478 V=800.0 PL=0
MOVL C01479 V=800.0 PL=0
MOVL C01480 V=800.0 PL=0
MOVL C01481 V=800.0 PL=0
MOVL C01482 V=800.0 PL=0
MOVL C01483 V=800.0 PL=0
MOVL C01484 V=800.0 PL=0
MOVL C01485 V=800.0 PL=0
MOVL C01486 V=800.0 PL=0
MOVL C01487 V=800.0 PL=0
MOVL C01488 V=800.0 PL=0
MOVL C01489 V=800.0 PL=0
MOVL C01490 V=800.0 PL=0
MOVL C01491 V=800.0 PL=0
MOVL C01492 V=800.0 PL=0
MOVL C01493 V=800.0 PL=0
MOVL C01494 V=800.0 PL=0
MOVL C01495 V=800.0 PL=0
MOVL C01496 V=800.0 PL=0
MOVL C01497 V=800.0 PL=0
MOVL C01498 V=800.0 PL=0
MOVL C01499 V=800.0 PL=0
MOVL C01500 V=800.0 PL=0
MOVL C01501 V=800.0 PL=0
MOVL C01502 V=800.0 PL=0
MOVL C01503 V=800.0 PL=0
MOVL C01504 V=800.0 PL=0
MOVL C01505 V=800.0 PL=0
MOVL C01506 V=800.0 PL=0
MOVL C01507 V=800.0 PL=0
MOVL C01508 V=800.0 PL=0
MOVL C01509 V=800.0 PL=0
MOVL C01510 V=800.0 PL=0
MOVL C01511 V=800.0 PL=0
MOVL C01512 V=800.0 PL=0
MOVL C01513 V=800.0 PL=0
MOVL C01514 V=800.0 PL=0
MOVL C01515 V=800.0 PL=0
MOVL C01516 V=800.0 PL=0
MOVL C01517 V=800.0 PL=0
MOVL C01518 V=800.0 PL=0
MOVL C01519 V=800.0 PL=0
MOVL C01520 V=800.0 PL=0
MOVL C01521 V=800.0 PL=0
MOVL C01522 V=800.0 PL=0
MOVL C01523 V=800.0 PL=0
MOVL C01524 V=800.0 PL=0
MOVL C01525 V=800.0 PL=0
MOVL C01526 V=800.0 PL=0
MOVL C01527 V=800.0 PL=0
MOVL C01528 V=800.0 PL=0
MOVL C01529 V=800.0 PL=0
MOVL C01530 V=800.0 PL=0
MOVL C01531 V=800.0 PL=0
MOVL C01532 V=800.0 PL=0
MOVL C01533 V=800.0 PL=0
MOVL C01534 V=800.0 PL=0
MOVL C01535 V=800.0 PL=0
MOVL C01536 V=800.0 PL=0
MOVL C01537 V=800.0 PL=0
MOVL C01538 V=800.0 PL=0
MOVL C01539 V=800.0 PL=0
MOVL C01540 V=800.0 PL=0
MOVL C01541 V=800.0 PL=0
MOVL C01542 V=800.0 PL=0
MOVL C01543 V=800.0 PL=0
MOVL C01544 V=800.0 PL=0
MOVL C01545 V=800.0 PL=0
MOVL C01546 V=800.0 PL=0
MOVL C01547 V=800.0 PL=0
MOVL C01548 V=800.0 PL=0
MOVL C01549 V=800.0 PL=0
MOVL C01550 V=800.0 PL=0
MOVL C01551 V=800.0 PL=0
MOVL C01552 V=800.0 PL=0
MOVL C01553 V=800.0 PL=0
MOVL C01554 V=800.0 PL=0
MOVL C01555 V=800.0 PL=0
MOVL C01556 V=800.0 PL=0
MOVL C01557 V=800.0 PL=0
MOVL C01558 V=800.0 PL=0
MOVL C01559 V=800.0 PL=0
MOVL C01560 V=800.0 PL=0
MOVL C01561 V=800.0 PL=0
MOVL C01562 V=800.0 PL=0
MOVL C01563 V=800.0 PL=0
MOVL C01564 V=800.0 PL=0
MOVL C01565 V=800.0 PL=0
MOVL C01566 V=800.0 PL=0
MOVL C01567 V=800.0 PL=0
MOVL C01568 V=800.0 PL=0
MOVL C01569 V=800.0 PL=0
MOVL C01570 V=800.0 PL=0
MOVL C01571 V=800.0 PL=0
MOVL C01572 V=800.0 PL=0
MOVL C01573 V=800.0 PL=0
MOVL C01574 V=800.0 PL=0
MOVL C01575 V=800.0 PL=0
MOVL C01576 V=800.0 PL=0
MOVL C01577 V=800.0 PL=0
MOVL C01578 V=800.0 PL=0
MOVL C01579 V=800.0 PL=0
MOVL C01580 V=800.0 PL=0
MOVL C01581 V=800.0 PL=0
MOVL C01582 V=800.0 PL=0
MOVL C01583 V=800.0 PL=0
MOVL C01584 V=800.0 PL=0
MOVL C01585 V=800.0 PL=0
MOVL C01586 V=800.0 PL=0
MOVL C01587 V=800.0 PL=0
MOVL C01588 V=800.0 PL=0
MOVL C01589 V=800.0 PL=0
MOVL C01590 V=800.0 PL=0
MOVL C01591 V=800.0 PL=0
MOVL C01592 V=800.0 PL=0
MOVL C01593 V=800.0 PL=0
MOVL C01594 V=800.0 PL=0
MOVL C01595 V=800.0 PL=0
MOVL C01596 V=800.0 PL=0
MOVL C01597 V=800.0 PL=0
MOVL C01598 V=800.0 PL=0
MOVL C01599 V=800.0 PL=0
MOVL C01600 V=800.0 PL=0
MOVL C01601 V=800.0 PL=0
MOVL C01602 V=800.0 PL=0
MOVL C01603 V=800.0 PL=0
MOVL C01604 V=800.0 PL=0
MOVL C01605 V=800.0 PL=0
MOVL C01606 V=800.0 PL=0
MOVL C01607 V=800.0 PL=0
MOVL C01608 V=800.0 PL=0
MOVL C01609 V=800.0 PL=0
MOVL C01610 V=800.0 PL=0
MOVL C01611 V=800.0 PL=0
MOVL C01612 V=800.0 PL=0
MOVL C01613 V=800.0 PL=0
MOVL C01614 V=800.0 PL=0
MOVL C01615 V=800.0 PL=0
MOVL C01616 V=800.0 PL=0
MOVL C01617 V=800.0 PL=0
MOVL C01618 V=800.0 PL=0
MOVL C01619 V=800.0 PL=0
MOVL C01620 V=800.0 PL=0
MOVL C01621 V=800.0 PL=0
MOVL C01622 V=800.0 PL=0
MOVL C01623 V=800.0 PL=0
MOVL C01624 V=800.0 PL=0
MOVL C01625 V=800.0 PL=0
